    // ---- l0_silu: SILU ----
    v1[0] := v0[0] / (1.0 + EXP(-v0[0]));
    v1[1] := v0[1] / (1.0 + EXP(-v0[1]));
    v1[2] := v0[2] / (1.0 + EXP(-v0[2]));
    v1[3] := v0[3] / (1.0 + EXP(-v0[3]));
    v1[4] := v0[4] / (1.0 + EXP(-v0[4]));
    v1[5] := v0[5] / (1.0 + EXP(-v0[5]));
    v1[6] := v0[6] / (1.0 + EXP(-v0[6]));
    v1[7] := v0[7] / (1.0 + EXP(-v0[7]));
    v1[8] := v0[8] / (1.0 + EXP(-v0[8]));
    v1[9] := v0[9] / (1.0 + EXP(-v0[9]));
    v1[10] := v0[10] / (1.0 + EXP(-v0[10]));
    v1[11] := v0[11] / (1.0 + EXP(-v0[11]));
    v1[12] := v0[12] / (1.0 + EXP(-v0[12]));
    v1[13] := v0[13] / (1.0 + EXP(-v0[13]));
    v1[14] := v0[14] / (1.0 + EXP(-v0[14]));
    v1[15] := v0[15] / (1.0 + EXP(-v0[15]));
    v1[16] := v0[16] / (1.0 + EXP(-v0[16]));
    v1[17] := v0[17] / (1.0 + EXP(-v0[17]));
    v1[18] := v0[18] / (1.0 + EXP(-v0[18]));
    v1[19] := v0[19] / (1.0 + EXP(-v0[19]));
    v1[20] := v0[20] / (1.0 + EXP(-v0[20]));
    v1[21] := v0[21] / (1.0 + EXP(-v0[21]));
    v1[22] := v0[22] / (1.0 + EXP(-v0[22]));
    v1[23] := v0[23] / (1.0 + EXP(-v0[23]));
    v1[24] := v0[24] / (1.0 + EXP(-v0[24]));
    v1[25] := v0[25] / (1.0 + EXP(-v0[25]));
    v1[26] := v0[26] / (1.0 + EXP(-v0[26]));
    v1[27] := v0[27] / (1.0 + EXP(-v0[27]));

    // ---- l0_bspline: BsplineLUT(28x16, 15pts) HOISTED ----
    // Binary search ONCE per input, shared across outputs
    // --- Input 0: binary search ---
    lo := 0; hi := 14;
    WHILE hi - lo > 1 DO
        mid := lo + (hi - lo) / 2;
        IF v0[0] > "NeuroPLC_Weights".w0[mid] THEN lo := mid; ELSE hi := mid; END_IF;
    END_WHILE;
    t_val := (v0[0] - "NeuroPLC_Weights".w0[lo]) / ("NeuroPLC_Weights".w0[hi] - "NeuroPLC_Weights".w0[lo] + 1.0E-10);
    v3[0, 0] := "NeuroPLC_Weights".w1[0 + lo] * (1.0 - t_val) + "NeuroPLC_Weights".w1[0 + hi] * t_val;
    v3[1, 0] := "NeuroPLC_Weights".w1[420 + lo] * (1.0 - t_val) + "NeuroPLC_Weights".w1[420 + hi] * t_val;
    v3[2, 0] := "NeuroPLC_Weights".w1[840 + lo] * (1.0 - t_val) + "NeuroPLC_Weights".w1[840 + hi] * t_val;
    v3[3, 0] := "NeuroPLC_Weights".w1[1260 + lo] * (1.0 - t_val) + "NeuroPLC_Weights".w1[1260 + hi] * t_val;
    v3[4, 0] := "NeuroPLC_Weights".w1[1680 + lo] * (1.0 - t_val) + "NeuroPLC_Weights".w1[1680 + hi] * t_val;
    v3[5, 0] := "NeuroPLC_Weights".w1[2100 + lo] * (1.0 - t_val) + "NeuroPLC_Weights".w1[2100 + hi] * t_val;
    v3[6, 0] := "NeuroPLC_Weights".w1[2520 + lo] * (1.0 - t_val) + "NeuroPLC_Weights".w1[2520 + hi] * t_val;
    v3[7, 0] := "NeuroPLC_Weights".w1[2940 + lo] * (1.0 - t_val) + "NeuroPLC_Weights".w1[2940 + hi] * t_val;
    v3[8, 0] := "NeuroPLC_Weights".w1[3360 + lo] * (1.0 - t_val) + "NeuroPLC_Weights".w1[3360 + hi] * t_val;
    v3[9, 0] := "NeuroPLC_Weights".w1[3780 + lo] * (1.0 - t_val) + "NeuroPLC_Weights".w1[3780 + hi] * t_val;
    v3[10, 0] := "NeuroPLC_Weights".w1[4200 + lo] * (1.0 - t_val) + "NeuroPLC_Weights".w1[4200 + hi] * t_val;
    v3[11, 0] := "NeuroPLC_Weights".w1[4620 + lo] * (1.0 - t_val) + "NeuroPLC_Weights".w1[4620 + hi] * t_val;
    v3[12, 0] := "NeuroPLC_Weights".w1[5040 + lo] * (1.0 - t_val) + "NeuroPLC_Weights".w1[5040 + hi] * t_val;
    v3[13, 0] := "NeuroPLC_Weights".w1[5460 + lo] * (1.0 - t_val) + "NeuroPLC_Weights".w1[5460 + hi] * t_val;
    v3[14, 0] := "NeuroPLC_Weights".w1[5880 + lo] * (1.0 - t_val) + "NeuroPLC_Weights".w1[5880 + hi] * t_val;
    v3[15, 0] := "NeuroPLC_Weights".w1[6300 + lo] * (1.0 - t_val) + "NeuroPLC_Weights".w1[6300 + hi] * t_val;

    // --- Input 1: binary search ---
    lo := 0; hi := 14;
    WHILE hi - lo > 1 DO
        mid := lo + (hi - lo) / 2;
        IF v0[1] > "NeuroPLC_Weights".w0[mid] THEN lo := mid; ELSE hi := mid; END_IF;
    END_WHILE;
    t_val := (v0[1] - "NeuroPLC_Weights".w0[lo]) / ("NeuroPLC_Weights".w0[hi] - "NeuroPLC_Weights".w0[lo] + 1.0E-10);
    v3[0, 1] := "NeuroPLC_Weights".w1[15 + lo] * (1.0 - t_val) + "NeuroPLC_Weights".w1[15 + hi] * t_val;
    v3[1, 1] := "NeuroPLC_Weights".w1[435 + lo] * (1.0 - t_val) + "NeuroPLC_Weights".w1[435 + hi] * t_val;
    v3[2, 1] := "NeuroPLC_Weights".w1[855 + lo] * (1.0 - t_val) + "NeuroPLC_Weights".w1[855 + hi] * t_val;
    v3[3, 1] := "NeuroPLC_Weights".w1[1275 + lo] * (1.0 - t_val) + "NeuroPLC_Weights".w1[1275 + hi] * t_val;
    v3[4, 1] := "NeuroPLC_Weights".w1[1695 + lo] * (1.0 - t_val) + "NeuroPLC_Weights".w1[1695 + hi] * t_val;
    v3[5, 1] := "NeuroPLC_Weights".w1[2115 + lo] * (1.0 - t_val) + "NeuroPLC_Weights".w1[2115 + hi] * t_val;
    v3[6, 1] := "NeuroPLC_Weights".w1[2535 + lo] * (1.0 - t_val) + "NeuroPLC_Weights".w1[2535 + hi] * t_val;
    v3[7, 1] := "NeuroPLC_Weights".w1[2955 + lo] * (1.0 - t_val) + "NeuroPLC_Weights".w1[2955 + hi] * t_val;
    v3[8, 1] := "NeuroPLC_Weights".w1[3375 + lo] * (1.0 - t_val) + "NeuroPLC_Weights".w1[3375 + hi] * t_val;
    v3[9, 1] := "NeuroPLC_Weights".w1[3795 + lo] * (1.0 - t_val) + "NeuroPLC_Weights".w1[3795 + hi] * t_val;
    v3[10, 1] := "NeuroPLC_Weights".w1[4215 + lo] * (1.0 - t_val) + "NeuroPLC_Weights".w1[4215 + hi] * t_val;
    v3[11, 1] := "NeuroPLC_Weights".w1[4635 + lo] * (1.0 - t_val) + "NeuroPLC_Weights".w1[4635 + hi] * t_val;
    v3[12, 1] := "NeuroPLC_Weights".w1[5055 + lo] * (1.0 - t_val) + "NeuroPLC_Weights".w1[5055 + hi] * t_val;
    v3[13, 1] := "NeuroPLC_Weights".w1[5475 + lo] * (1.0 - t_val) + "NeuroPLC_Weights".w1[5475 + hi] * t_val;
    v3[14, 1] := "NeuroPLC_Weights".w1[5895 + lo] * (1.0 - t_val) + "NeuroPLC_Weights".w1[5895 + hi] * t_val;
    v3[15, 1] := "NeuroPLC_Weights".w1[6315 + lo] * (1.0 - t_val) + "NeuroPLC_Weights".w1[6315 + hi] * t_val;

    // --- Input 2: binary search ---
    lo := 0; hi := 14;
    WHILE hi - lo > 1 DO
        mid := lo + (hi - lo) / 2;
        IF v0[2] > "NeuroPLC_Weights".w0[mid] THEN lo := mid; ELSE hi := mid; END_IF;
    END_WHILE;
    t_val := (v0[2] - "NeuroPLC_Weights".w0[lo]) / ("NeuroPLC_Weights".w0[hi] - "NeuroPLC_Weights".w0[lo] + 1.0E-10);
    v3[0, 2] := "NeuroPLC_Weights".w1[30 + lo] * (1.0 - t_val) + "NeuroPLC_Weights".w1[30 + hi] * t_val;
    v3[1, 2] := "NeuroPLC_Weights".w1[450 + lo] * (1.0 - t_val) + "NeuroPLC_Weights".w1[450 + hi] * t_val;
    v3[2, 2] := "NeuroPLC_Weights".w1[870 + lo] * (1.0 - t_val) + "NeuroPLC_Weights".w1[870 + hi] * t_val;
    v3[3, 2] := "NeuroPLC_Weights".w1[1290 + lo] * (1.0 - t_val) + "NeuroPLC_Weights".w1[1290 + hi] * t_val;
    v3[4, 2] := "NeuroPLC_Weights".w1[1710 + lo] * (1.0 - t_val) + "NeuroPLC_Weights".w1[1710 + hi] * t_val;
    v3[5, 2] := "NeuroPLC_Weights".w1[2130 + lo] * (1.0 - t_val) + "NeuroPLC_Weights".w1[2130 + hi] * t_val;
    v3[6, 2] := "NeuroPLC_Weights".w1[2550 + lo] * (1.0 - t_val) + "NeuroPLC_Weights".w1[2550 + hi] * t_val;
    v3[7, 2] := "NeuroPLC_Weights".w1[2970 + lo] * (1.0 - t_val) + "NeuroPLC_Weights".w1[2970 + hi] * t_val;
    v3[8, 2] := "NeuroPLC_Weights".w1[3390 + lo] * (1.0 - t_val) + "NeuroPLC_Weights".w1[3390 + hi] * t_val;
    v3[9, 2] := "NeuroPLC_Weights".w1[3810 + lo] * (1.0 - t_val) + "NeuroPLC_Weights".w1[3810 + hi] * t_val;
    v3[10, 2] := "NeuroPLC_Weights".w1[4230 + lo] * (1.0 - t_val) + "NeuroPLC_Weights".w1[4230 + hi] * t_val;
    v3[11, 2] := "NeuroPLC_Weights".w1[4650 + lo] * (1.0 - t_val) + "NeuroPLC_Weights".w1[4650 + hi] * t_val;
    v3[12, 2] := "NeuroPLC_Weights".w1[5070 + lo] * (1.0 - t_val) + "NeuroPLC_Weights".w1[5070 + hi] * t_val;
    v3[13, 2] := "NeuroPLC_Weights".w1[5490 + lo] * (1.0 - t_val) + "NeuroPLC_Weights".w1[5490 + hi] * t_val;
    v3[14, 2] := "NeuroPLC_Weights".w1[5910 + lo] * (1.0 - t_val) + "NeuroPLC_Weights".w1[5910 + hi] * t_val;
    v3[15, 2] := "NeuroPLC_Weights".w1[6330 + lo] * (1.0 - t_val) + "NeuroPLC_Weights".w1[6330 + hi] * t_val;

    // --- Input 3: binary search ---
    lo := 0; hi := 14;
    WHILE hi - lo > 1 DO
        mid := lo + (hi - lo) / 2;
        IF v0[3] > "NeuroPLC_Weights".w0[mid] THEN lo := mid; ELSE hi := mid; END_IF;
    END_WHILE;
    t_val := (v0[3] - "NeuroPLC_Weights".w0[lo]) / ("NeuroPLC_Weights".w0[hi] - "NeuroPLC_Weights".w0[lo] + 1.0E-10);
    v3[0, 3] := "NeuroPLC_Weights".w1[45 + lo] * (1.0 - t_val) + "NeuroPLC_Weights".w1[45 + hi] * t_val;
    v3[1, 3] := "NeuroPLC_Weights".w1[465 + lo] * (1.0 - t_val) + "NeuroPLC_Weights".w1[465 + hi] * t_val;
    v3[2, 3] := "NeuroPLC_Weights".w1[885 + lo] * (1.0 - t_val) + "NeuroPLC_Weights".w1[885 + hi] * t_val;
    v3[3, 3] := "NeuroPLC_Weights".w1[1305 + lo] * (1.0 - t_val) + "NeuroPLC_Weights".w1[1305 + hi] * t_val;
    v3[4, 3] := "NeuroPLC_Weights".w1[1725 + lo] * (1.0 - t_val) + "NeuroPLC_Weights".w1[1725 + hi] * t_val;
    v3[5, 3] := "NeuroPLC_Weights".w1[2145 + lo] * (1.0 - t_val) + "NeuroPLC_Weights".w1[2145 + hi] * t_val;
    v3[6, 3] := "NeuroPLC_Weights".w1[2565 + lo] * (1.0 - t_val) + "NeuroPLC_Weights".w1[2565 + hi] * t_val;
    v3[7, 3] := "NeuroPLC_Weights".w1[2985 + lo] * (1.0 - t_val) + "NeuroPLC_Weights".w1[2985 + hi] * t_val;
    v3[8, 3] := "NeuroPLC_Weights".w1[3405 + lo] * (1.0 - t_val) + "NeuroPLC_Weights".w1[3405 + hi] * t_val;
    v3[9, 3] := "NeuroPLC_Weights".w1[3825 + lo] * (1.0 - t_val) + "NeuroPLC_Weights".w1[3825 + hi] * t_val;
    v3[10, 3] := "NeuroPLC_Weights".w1[4245 + lo] * (1.0 - t_val) + "NeuroPLC_Weights".w1[4245 + hi] * t_val;
    v3[11, 3] := "NeuroPLC_Weights".w1[4665 + lo] * (1.0 - t_val) + "NeuroPLC_Weights".w1[4665 + hi] * t_val;
    v3[12, 3] := "NeuroPLC_Weights".w1[5085 + lo] * (1.0 - t_val) + "NeuroPLC_Weights".w1[5085 + hi] * t_val;
    v3[13, 3] := "NeuroPLC_Weights".w1[5505 + lo] * (1.0 - t_val) + "NeuroPLC_Weights".w1[5505 + hi] * t_val;
    v3[14, 3] := "NeuroPLC_Weights".w1[5925 + lo] * (1.0 - t_val) + "NeuroPLC_Weights".w1[5925 + hi] * t_val;
    v3[15, 3] := "NeuroPLC_Weights".w1[6345 + lo] * (1.0 - t_val) + "NeuroPLC_Weights".w1[6345 + hi] * t_val;

    // --- Input 4: binary search ---
    lo := 0; hi := 14;
    WHILE hi - lo > 1 DO
        mid := lo + (hi - lo) / 2;
        IF v0[4] > "NeuroPLC_Weights".w0[mid] THEN lo := mid; ELSE hi := mid; END_IF;
    END_WHILE;
    t_val := (v0[4] - "NeuroPLC_Weights".w0[lo]) / ("NeuroPLC_Weights".w0[hi] - "NeuroPLC_Weights".w0[lo] + 1.0E-10);
    v3[0, 4] := "NeuroPLC_Weights".w1[60 + lo] * (1.0 - t_val) + "NeuroPLC_Weights".w1[60 + hi] * t_val;
    v3[1, 4] := "NeuroPLC_Weights".w1[480 + lo] * (1.0 - t_val) + "NeuroPLC_Weights".w1[480 + hi] * t_val;
    v3[2, 4] := "NeuroPLC_Weights".w1[900 + lo] * (1.0 - t_val) + "NeuroPLC_Weights".w1[900 + hi] * t_val;
    v3[3, 4] := "NeuroPLC_Weights".w1[1320 + lo] * (1.0 - t_val) + "NeuroPLC_Weights".w1[1320 + hi] * t_val;
    v3[4, 4] := "NeuroPLC_Weights".w1[1740 + lo] * (1.0 - t_val) + "NeuroPLC_Weights".w1[1740 + hi] * t_val;
    v3[5, 4] := "NeuroPLC_Weights".w1[2160 + lo] * (1.0 - t_val) + "NeuroPLC_Weights".w1[2160 + hi] * t_val;
    v3[6, 4] := "NeuroPLC_Weights".w1[2580 + lo] * (1.0 - t_val) + "NeuroPLC_Weights".w1[2580 + hi] * t_val;
    v3[7, 4] := "NeuroPLC_Weights".w1[3000 + lo] * (1.0 - t_val) + "NeuroPLC_Weights".w1[3000 + hi] * t_val;
    v3[8, 4] := "NeuroPLC_Weights".w1[3420 + lo] * (1.0 - t_val) + "NeuroPLC_Weights".w1[3420 + hi] * t_val;
    v3[9, 4] := "NeuroPLC_Weights".w1[3840 + lo] * (1.0 - t_val) + "NeuroPLC_Weights".w1[3840 + hi] * t_val;
    v3[10, 4] := "NeuroPLC_Weights".w1[4260 + lo] * (1.0 - t_val) + "NeuroPLC_Weights".w1[4260 + hi] * t_val;
    v3[11, 4] := "NeuroPLC_Weights".w1[4680 + lo] * (1.0 - t_val) + "NeuroPLC_Weights".w1[4680 + hi] * t_val;
    v3[12, 4] := "NeuroPLC_Weights".w1[5100 + lo] * (1.0 - t_val) + "NeuroPLC_Weights".w1[5100 + hi] * t_val;
    v3[13, 4] := "NeuroPLC_Weights".w1[5520 + lo] * (1.0 - t_val) + "NeuroPLC_Weights".w1[5520 + hi] * t_val;
    v3[14, 4] := "NeuroPLC_Weights".w1[5940 + lo] * (1.0 - t_val) + "NeuroPLC_Weights".w1[5940 + hi] * t_val;
    v3[15, 4] := "NeuroPLC_Weights".w1[6360 + lo] * (1.0 - t_val) + "NeuroPLC_Weights".w1[6360 + hi] * t_val;

    // --- Input 5: binary search ---
    lo := 0; hi := 14;
    WHILE hi - lo > 1 DO
        mid := lo + (hi - lo) / 2;
        IF v0[5] > "NeuroPLC_Weights".w0[mid] THEN lo := mid; ELSE hi := mid; END_IF;
    END_WHILE;
    t_val := (v0[5] - "NeuroPLC_Weights".w0[lo]) / ("NeuroPLC_Weights".w0[hi] - "NeuroPLC_Weights".w0[lo] + 1.0E-10);
    v3[0, 5] := "NeuroPLC_Weights".w1[75 + lo] * (1.0 - t_val) + "NeuroPLC_Weights".w1[75 + hi] * t_val;
    v3[1, 5] := "NeuroPLC_Weights".w1[495 + lo] * (1.0 - t_val) + "NeuroPLC_Weights".w1[495 + hi] * t_val;
    v3[2, 5] := "NeuroPLC_Weights".w1[915 + lo] * (1.0 - t_val) + "NeuroPLC_Weights".w1[915 + hi] * t_val;
    v3[3, 5] := "NeuroPLC_Weights".w1[1335 + lo] * (1.0 - t_val) + "NeuroPLC_Weights".w1[1335 + hi] * t_val;
    v3[4, 5] := "NeuroPLC_Weights".w1[1755 + lo] * (1.0 - t_val) + "NeuroPLC_Weights".w1[1755 + hi] * t_val;
    v3[5, 5] := "NeuroPLC_Weights".w1[2175 + lo] * (1.0 - t_val) + "NeuroPLC_Weights".w1[2175 + hi] * t_val;
    v3[6, 5] := "NeuroPLC_Weights".w1[2595 + lo] * (1.0 - t_val) + "NeuroPLC_Weights".w1[2595 + hi] * t_val;
    v3[7, 5] := "NeuroPLC_Weights".w1[3015 + lo] * (1.0 - t_val) + "NeuroPLC_Weights".w1[3015 + hi] * t_val;
    v3[8, 5] := "NeuroPLC_Weights".w1[3435 + lo] * (1.0 - t_val) + "NeuroPLC_Weights".w1[3435 + hi] * t_val;
    v3[9, 5] := "NeuroPLC_Weights".w1[3855 + lo] * (1.0 - t_val) + "NeuroPLC_Weights".w1[3855 + hi] * t_val;
    v3[10, 5] := "NeuroPLC_Weights".w1[4275 + lo] * (1.0 - t_val) + "NeuroPLC_Weights".w1[4275 + hi] * t_val;
    v3[11, 5] := "NeuroPLC_Weights".w1[4695 + lo] * (1.0 - t_val) + "NeuroPLC_Weights".w1[4695 + hi] * t_val;
    v3[12, 5] := "NeuroPLC_Weights".w1[5115 + lo] * (1.0 - t_val) + "NeuroPLC_Weights".w1[5115 + hi] * t_val;
    v3[13, 5] := "NeuroPLC_Weights".w1[5535 + lo] * (1.0 - t_val) + "NeuroPLC_Weights".w1[5535 + hi] * t_val;
    v3[14, 5] := "NeuroPLC_Weights".w1[5955 + lo] * (1.0 - t_val) + "NeuroPLC_Weights".w1[5955 + hi] * t_val;
    v3[15, 5] := "NeuroPLC_Weights".w1[6375 + lo] * (1.0 - t_val) + "NeuroPLC_Weights".w1[6375 + hi] * t_val;

    // --- Input 6: binary search ---
    lo := 0; hi := 14;
    WHILE hi - lo > 1 DO
        mid := lo + (hi - lo) / 2;
        IF v0[6] > "NeuroPLC_Weights".w0[mid] THEN lo := mid; ELSE hi := mid; END_IF;
    END_WHILE;
    t_val := (v0[6] - "NeuroPLC_Weights".w0[lo]) / ("NeuroPLC_Weights".w0[hi] - "NeuroPLC_Weights".w0[lo] + 1.0E-10);
    v3[0, 6] := "NeuroPLC_Weights".w1[90 + lo] * (1.0 - t_val) + "NeuroPLC_Weights".w1[90 + hi] * t_val;
    v3[1, 6] := "NeuroPLC_Weights".w1[510 + lo] * (1.0 - t_val) + "NeuroPLC_Weights".w1[510 + hi] * t_val;
    v3[2, 6] := "NeuroPLC_Weights".w1[930 + lo] * (1.0 - t_val) + "NeuroPLC_Weights".w1[930 + hi] * t_val;
    v3[3, 6] := "NeuroPLC_Weights".w1[1350 + lo] * (1.0 - t_val) + "NeuroPLC_Weights".w1[1350 + hi] * t_val;
    v3[4, 6] := "NeuroPLC_Weights".w1[1770 + lo] * (1.0 - t_val) + "NeuroPLC_Weights".w1[1770 + hi] * t_val;
    v3[5, 6] := "NeuroPLC_Weights".w1[2190 + lo] * (1.0 - t_val) + "NeuroPLC_Weights".w1[2190 + hi] * t_val;
    v3[6, 6] := "NeuroPLC_Weights".w1[2610 + lo] * (1.0 - t_val) + "NeuroPLC_Weights".w1[2610 + hi] * t_val;
    v3[7, 6] := "NeuroPLC_Weights".w1[3030 + lo] * (1.0 - t_val) + "NeuroPLC_Weights".w1[3030 + hi] * t_val;
    v3[8, 6] := "NeuroPLC_Weights".w1[3450 + lo] * (1.0 - t_val) + "NeuroPLC_Weights".w1[3450 + hi] * t_val;
    v3[9, 6] := "NeuroPLC_Weights".w1[3870 + lo] * (1.0 - t_val) + "NeuroPLC_Weights".w1[3870 + hi] * t_val;
    v3[10, 6] := "NeuroPLC_Weights".w1[4290 + lo] * (1.0 - t_val) + "NeuroPLC_Weights".w1[4290 + hi] * t_val;
    v3[11, 6] := "NeuroPLC_Weights".w1[4710 + lo] * (1.0 - t_val) + "NeuroPLC_Weights".w1[4710 + hi] * t_val;
    v3[12, 6] := "NeuroPLC_Weights".w1[5130 + lo] * (1.0 - t_val) + "NeuroPLC_Weights".w1[5130 + hi] * t_val;
    v3[13, 6] := "NeuroPLC_Weights".w1[5550 + lo] * (1.0 - t_val) + "NeuroPLC_Weights".w1[5550 + hi] * t_val;
    v3[14, 6] := "NeuroPLC_Weights".w1[5970 + lo] * (1.0 - t_val) + "NeuroPLC_Weights".w1[5970 + hi] * t_val;
    v3[15, 6] := "NeuroPLC_Weights".w1[6390 + lo] * (1.0 - t_val) + "NeuroPLC_Weights".w1[6390 + hi] * t_val;

    // --- Input 7: binary search ---
    lo := 0; hi := 14;
    WHILE hi - lo > 1 DO
        mid := lo + (hi - lo) / 2;
        IF v0[7] > "NeuroPLC_Weights".w0[mid] THEN lo := mid; ELSE hi := mid; END_IF;
    END_WHILE;
    t_val := (v0[7] - "NeuroPLC_Weights".w0[lo]) / ("NeuroPLC_Weights".w0[hi] - "NeuroPLC_Weights".w0[lo] + 1.0E-10);
    v3[0, 7] := "NeuroPLC_Weights".w1[105 + lo] * (1.0 - t_val) + "NeuroPLC_Weights".w1[105 + hi] * t_val;
    v3[1, 7] := "NeuroPLC_Weights".w1[525 + lo] * (1.0 - t_val) + "NeuroPLC_Weights".w1[525 + hi] * t_val;
    v3[2, 7] := "NeuroPLC_Weights".w1[945 + lo] * (1.0 - t_val) + "NeuroPLC_Weights".w1[945 + hi] * t_val;
    v3[3, 7] := "NeuroPLC_Weights".w1[1365 + lo] * (1.0 - t_val) + "NeuroPLC_Weights".w1[1365 + hi] * t_val;
    v3[4, 7] := "NeuroPLC_Weights".w1[1785 + lo] * (1.0 - t_val) + "NeuroPLC_Weights".w1[1785 + hi] * t_val;
    v3[5, 7] := "NeuroPLC_Weights".w1[2205 + lo] * (1.0 - t_val) + "NeuroPLC_Weights".w1[2205 + hi] * t_val;
    v3[6, 7] := "NeuroPLC_Weights".w1[2625 + lo] * (1.0 - t_val) + "NeuroPLC_Weights".w1[2625 + hi] * t_val;
    v3[7, 7] := "NeuroPLC_Weights".w1[3045 + lo] * (1.0 - t_val) + "NeuroPLC_Weights".w1[3045 + hi] * t_val;
    v3[8, 7] := "NeuroPLC_Weights".w1[3465 + lo] * (1.0 - t_val) + "NeuroPLC_Weights".w1[3465 + hi] * t_val;
    v3[9, 7] := "NeuroPLC_Weights".w1[3885 + lo] * (1.0 - t_val) + "NeuroPLC_Weights".w1[3885 + hi] * t_val;
    v3[10, 7] := "NeuroPLC_Weights".w1[4305 + lo] * (1.0 - t_val) + "NeuroPLC_Weights".w1[4305 + hi] * t_val;
    v3[11, 7] := "NeuroPLC_Weights".w1[4725 + lo] * (1.0 - t_val) + "NeuroPLC_Weights".w1[4725 + hi] * t_val;
    v3[12, 7] := "NeuroPLC_Weights".w1[5145 + lo] * (1.0 - t_val) + "NeuroPLC_Weights".w1[5145 + hi] * t_val;
    v3[13, 7] := "NeuroPLC_Weights".w1[5565 + lo] * (1.0 - t_val) + "NeuroPLC_Weights".w1[5565 + hi] * t_val;
    v3[14, 7] := "NeuroPLC_Weights".w1[5985 + lo] * (1.0 - t_val) + "NeuroPLC_Weights".w1[5985 + hi] * t_val;
    v3[15, 7] := "NeuroPLC_Weights".w1[6405 + lo] * (1.0 - t_val) + "NeuroPLC_Weights".w1[6405 + hi] * t_val;

    // --- Input 8: binary search ---
    lo := 0; hi := 14;
    WHILE hi - lo > 1 DO
        mid := lo + (hi - lo) / 2;
        IF v0[8] > "NeuroPLC_Weights".w0[mid] THEN lo := mid; ELSE hi := mid; END_IF;
    END_WHILE;
    t_val := (v0[8] - "NeuroPLC_Weights".w0[lo]) / ("NeuroPLC_Weights".w0[hi] - "NeuroPLC_Weights".w0[lo] + 1.0E-10);
    v3[0, 8] := "NeuroPLC_Weights".w1[120 + lo] * (1.0 - t_val) + "NeuroPLC_Weights".w1[120 + hi] * t_val;
    v3[1, 8] := "NeuroPLC_Weights".w1[540 + lo] * (1.0 - t_val) + "NeuroPLC_Weights".w1[540 + hi] * t_val;
    v3[2, 8] := "NeuroPLC_Weights".w1[960 + lo] * (1.0 - t_val) + "NeuroPLC_Weights".w1[960 + hi] * t_val;
    v3[3, 8] := "NeuroPLC_Weights".w1[1380 + lo] * (1.0 - t_val) + "NeuroPLC_Weights".w1[1380 + hi] * t_val;
    v3[4, 8] := "NeuroPLC_Weights".w1[1800 + lo] * (1.0 - t_val) + "NeuroPLC_Weights".w1[1800 + hi] * t_val;
    v3[5, 8] := "NeuroPLC_Weights".w1[2220 + lo] * (1.0 - t_val) + "NeuroPLC_Weights".w1[2220 + hi] * t_val;
    v3[6, 8] := "NeuroPLC_Weights".w1[2640 + lo] * (1.0 - t_val) + "NeuroPLC_Weights".w1[2640 + hi] * t_val;
    v3[7, 8] := "NeuroPLC_Weights".w1[3060 + lo] * (1.0 - t_val) + "NeuroPLC_Weights".w1[3060 + hi] * t_val;
    v3[8, 8] := "NeuroPLC_Weights".w1[3480 + lo] * (1.0 - t_val) + "NeuroPLC_Weights".w1[3480 + hi] * t_val;
    v3[9, 8] := "NeuroPLC_Weights".w1[3900 + lo] * (1.0 - t_val) + "NeuroPLC_Weights".w1[3900 + hi] * t_val;
    v3[10, 8] := "NeuroPLC_Weights".w1[4320 + lo] * (1.0 - t_val) + "NeuroPLC_Weights".w1[4320 + hi] * t_val;
    v3[11, 8] := "NeuroPLC_Weights".w1[4740 + lo] * (1.0 - t_val) + "NeuroPLC_Weights".w1[4740 + hi] * t_val;
    v3[12, 8] := "NeuroPLC_Weights".w1[5160 + lo] * (1.0 - t_val) + "NeuroPLC_Weights".w1[5160 + hi] * t_val;
    v3[13, 8] := "NeuroPLC_Weights".w1[5580 + lo] * (1.0 - t_val) + "NeuroPLC_Weights".w1[5580 + hi] * t_val;
    v3[14, 8] := "NeuroPLC_Weights".w1[6000 + lo] * (1.0 - t_val) + "NeuroPLC_Weights".w1[6000 + hi] * t_val;
    v3[15, 8] := "NeuroPLC_Weights".w1[6420 + lo] * (1.0 - t_val) + "NeuroPLC_Weights".w1[6420 + hi] * t_val;

    // --- Input 9: binary search ---
    lo := 0; hi := 14;
    WHILE hi - lo > 1 DO
        mid := lo + (hi - lo) / 2;
        IF v0[9] > "NeuroPLC_Weights".w0[mid] THEN lo := mid; ELSE hi := mid; END_IF;
    END_WHILE;
    t_val := (v0[9] - "NeuroPLC_Weights".w0[lo]) / ("NeuroPLC_Weights".w0[hi] - "NeuroPLC_Weights".w0[lo] + 1.0E-10);
    v3[0, 9] := "NeuroPLC_Weights".w1[135 + lo] * (1.0 - t_val) + "NeuroPLC_Weights".w1[135 + hi] * t_val;
    v3[1, 9] := "NeuroPLC_Weights".w1[555 + lo] * (1.0 - t_val) + "NeuroPLC_Weights".w1[555 + hi] * t_val;
    v3[2, 9] := "NeuroPLC_Weights".w1[975 + lo] * (1.0 - t_val) + "NeuroPLC_Weights".w1[975 + hi] * t_val;
    v3[3, 9] := "NeuroPLC_Weights".w1[1395 + lo] * (1.0 - t_val) + "NeuroPLC_Weights".w1[1395 + hi] * t_val;
    v3[4, 9] := "NeuroPLC_Weights".w1[1815 + lo] * (1.0 - t_val) + "NeuroPLC_Weights".w1[1815 + hi] * t_val;
    v3[5, 9] := "NeuroPLC_Weights".w1[2235 + lo] * (1.0 - t_val) + "NeuroPLC_Weights".w1[2235 + hi] * t_val;
    v3[6, 9] := "NeuroPLC_Weights".w1[2655 + lo] * (1.0 - t_val) + "NeuroPLC_Weights".w1[2655 + hi] * t_val;
    v3[7, 9] := "NeuroPLC_Weights".w1[3075 + lo] * (1.0 - t_val) + "NeuroPLC_Weights".w1[3075 + hi] * t_val;
    v3[8, 9] := "NeuroPLC_Weights".w1[3495 + lo] * (1.0 - t_val) + "NeuroPLC_Weights".w1[3495 + hi] * t_val;
    v3[9, 9] := "NeuroPLC_Weights".w1[3915 + lo] * (1.0 - t_val) + "NeuroPLC_Weights".w1[3915 + hi] * t_val;
    v3[10, 9] := "NeuroPLC_Weights".w1[4335 + lo] * (1.0 - t_val) + "NeuroPLC_Weights".w1[4335 + hi] * t_val;
    v3[11, 9] := "NeuroPLC_Weights".w1[4755 + lo] * (1.0 - t_val) + "NeuroPLC_Weights".w1[4755 + hi] * t_val;
    v3[12, 9] := "NeuroPLC_Weights".w1[5175 + lo] * (1.0 - t_val) + "NeuroPLC_Weights".w1[5175 + hi] * t_val;
    v3[13, 9] := "NeuroPLC_Weights".w1[5595 + lo] * (1.0 - t_val) + "NeuroPLC_Weights".w1[5595 + hi] * t_val;
    v3[14, 9] := "NeuroPLC_Weights".w1[6015 + lo] * (1.0 - t_val) + "NeuroPLC_Weights".w1[6015 + hi] * t_val;
    v3[15, 9] := "NeuroPLC_Weights".w1[6435 + lo] * (1.0 - t_val) + "NeuroPLC_Weights".w1[6435 + hi] * t_val;

    // --- Input 10: binary search ---
    lo := 0; hi := 14;
    WHILE hi - lo > 1 DO
        mid := lo + (hi - lo) / 2;
        IF v0[10] > "NeuroPLC_Weights".w0[mid] THEN lo := mid; ELSE hi := mid; END_IF;
    END_WHILE;
    t_val := (v0[10] - "NeuroPLC_Weights".w0[lo]) / ("NeuroPLC_Weights".w0[hi] - "NeuroPLC_Weights".w0[lo] + 1.0E-10);
    v3[0, 10] := "NeuroPLC_Weights".w1[150 + lo] * (1.0 - t_val) + "NeuroPLC_Weights".w1[150 + hi] * t_val;
    v3[1, 10] := "NeuroPLC_Weights".w1[570 + lo] * (1.0 - t_val) + "NeuroPLC_Weights".w1[570 + hi] * t_val;
    v3[2, 10] := "NeuroPLC_Weights".w1[990 + lo] * (1.0 - t_val) + "NeuroPLC_Weights".w1[990 + hi] * t_val;
    v3[3, 10] := "NeuroPLC_Weights".w1[1410 + lo] * (1.0 - t_val) + "NeuroPLC_Weights".w1[1410 + hi] * t_val;
    v3[4, 10] := "NeuroPLC_Weights".w1[1830 + lo] * (1.0 - t_val) + "NeuroPLC_Weights".w1[1830 + hi] * t_val;
    v3[5, 10] := "NeuroPLC_Weights".w1[2250 + lo] * (1.0 - t_val) + "NeuroPLC_Weights".w1[2250 + hi] * t_val;
    v3[6, 10] := "NeuroPLC_Weights".w1[2670 + lo] * (1.0 - t_val) + "NeuroPLC_Weights".w1[2670 + hi] * t_val;
    v3[7, 10] := "NeuroPLC_Weights".w1[3090 + lo] * (1.0 - t_val) + "NeuroPLC_Weights".w1[3090 + hi] * t_val;
    v3[8, 10] := "NeuroPLC_Weights".w1[3510 + lo] * (1.0 - t_val) + "NeuroPLC_Weights".w1[3510 + hi] * t_val;
    v3[9, 10] := "NeuroPLC_Weights".w1[3930 + lo] * (1.0 - t_val) + "NeuroPLC_Weights".w1[3930 + hi] * t_val;
    v3[10, 10] := "NeuroPLC_Weights".w1[4350 + lo] * (1.0 - t_val) + "NeuroPLC_Weights".w1[4350 + hi] * t_val;
    v3[11, 10] := "NeuroPLC_Weights".w1[4770 + lo] * (1.0 - t_val) + "NeuroPLC_Weights".w1[4770 + hi] * t_val;
    v3[12, 10] := "NeuroPLC_Weights".w1[5190 + lo] * (1.0 - t_val) + "NeuroPLC_Weights".w1[5190 + hi] * t_val;
    v3[13, 10] := "NeuroPLC_Weights".w1[5610 + lo] * (1.0 - t_val) + "NeuroPLC_Weights".w1[5610 + hi] * t_val;
    v3[14, 10] := "NeuroPLC_Weights".w1[6030 + lo] * (1.0 - t_val) + "NeuroPLC_Weights".w1[6030 + hi] * t_val;
    v3[15, 10] := "NeuroPLC_Weights".w1[6450 + lo] * (1.0 - t_val) + "NeuroPLC_Weights".w1[6450 + hi] * t_val;

    // --- Input 11: binary search ---
    lo := 0; hi := 14;
    WHILE hi - lo > 1 DO
        mid := lo + (hi - lo) / 2;
        IF v0[11] > "NeuroPLC_Weights".w0[mid] THEN lo := mid; ELSE hi := mid; END_IF;
    END_WHILE;
    t_val := (v0[11] - "NeuroPLC_Weights".w0[lo]) / ("NeuroPLC_Weights".w0[hi] - "NeuroPLC_Weights".w0[lo] + 1.0E-10);
    v3[0, 11] := "NeuroPLC_Weights".w1[165 + lo] * (1.0 - t_val) + "NeuroPLC_Weights".w1[165 + hi] * t_val;
    v3[1, 11] := "NeuroPLC_Weights".w1[585 + lo] * (1.0 - t_val) + "NeuroPLC_Weights".w1[585 + hi] * t_val;
    v3[2, 11] := "NeuroPLC_Weights".w1[1005 + lo] * (1.0 - t_val) + "NeuroPLC_Weights".w1[1005 + hi] * t_val;
    v3[3, 11] := "NeuroPLC_Weights".w1[1425 + lo] * (1.0 - t_val) + "NeuroPLC_Weights".w1[1425 + hi] * t_val;
    v3[4, 11] := "NeuroPLC_Weights".w1[1845 + lo] * (1.0 - t_val) + "NeuroPLC_Weights".w1[1845 + hi] * t_val;
    v3[5, 11] := "NeuroPLC_Weights".w1[2265 + lo] * (1.0 - t_val) + "NeuroPLC_Weights".w1[2265 + hi] * t_val;
    v3[6, 11] := "NeuroPLC_Weights".w1[2685 + lo] * (1.0 - t_val) + "NeuroPLC_Weights".w1[2685 + hi] * t_val;
    v3[7, 11] := "NeuroPLC_Weights".w1[3105 + lo] * (1.0 - t_val) + "NeuroPLC_Weights".w1[3105 + hi] * t_val;
    v3[8, 11] := "NeuroPLC_Weights".w1[3525 + lo] * (1.0 - t_val) + "NeuroPLC_Weights".w1[3525 + hi] * t_val;
    v3[9, 11] := "NeuroPLC_Weights".w1[3945 + lo] * (1.0 - t_val) + "NeuroPLC_Weights".w1[3945 + hi] * t_val;
    v3[10, 11] := "NeuroPLC_Weights".w1[4365 + lo] * (1.0 - t_val) + "NeuroPLC_Weights".w1[4365 + hi] * t_val;
    v3[11, 11] := "NeuroPLC_Weights".w1[4785 + lo] * (1.0 - t_val) + "NeuroPLC_Weights".w1[4785 + hi] * t_val;
    v3[12, 11] := "NeuroPLC_Weights".w1[5205 + lo] * (1.0 - t_val) + "NeuroPLC_Weights".w1[5205 + hi] * t_val;
    v3[13, 11] := "NeuroPLC_Weights".w1[5625 + lo] * (1.0 - t_val) + "NeuroPLC_Weights".w1[5625 + hi] * t_val;
    v3[14, 11] := "NeuroPLC_Weights".w1[6045 + lo] * (1.0 - t_val) + "NeuroPLC_Weights".w1[6045 + hi] * t_val;
    v3[15, 11] := "NeuroPLC_Weights".w1[6465 + lo] * (1.0 - t_val) + "NeuroPLC_Weights".w1[6465 + hi] * t_val;

    // --- Input 12: binary search ---
    lo := 0; hi := 14;
    WHILE hi - lo > 1 DO
        mid := lo + (hi - lo) / 2;
        IF v0[12] > "NeuroPLC_Weights".w0[mid] THEN lo := mid; ELSE hi := mid; END_IF;
    END_WHILE;
    t_val := (v0[12] - "NeuroPLC_Weights".w0[lo]) / ("NeuroPLC_Weights".w0[hi] - "NeuroPLC_Weights".w0[lo] + 1.0E-10);
    v3[0, 12] := "NeuroPLC_Weights".w1[180 + lo] * (1.0 - t_val) + "NeuroPLC_Weights".w1[180 + hi] * t_val;
    v3[1, 12] := "NeuroPLC_Weights".w1[600 + lo] * (1.0 - t_val) + "NeuroPLC_Weights".w1[600 + hi] * t_val;
    v3[2, 12] := "NeuroPLC_Weights".w1[1020 + lo] * (1.0 - t_val) + "NeuroPLC_Weights".w1[1020 + hi] * t_val;
    v3[3, 12] := "NeuroPLC_Weights".w1[1440 + lo] * (1.0 - t_val) + "NeuroPLC_Weights".w1[1440 + hi] * t_val;
    v3[4, 12] := "NeuroPLC_Weights".w1[1860 + lo] * (1.0 - t_val) + "NeuroPLC_Weights".w1[1860 + hi] * t_val;
    v3[5, 12] := "NeuroPLC_Weights".w1[2280 + lo] * (1.0 - t_val) + "NeuroPLC_Weights".w1[2280 + hi] * t_val;
    v3[6, 12] := "NeuroPLC_Weights".w1[2700 + lo] * (1.0 - t_val) + "NeuroPLC_Weights".w1[2700 + hi] * t_val;
    v3[7, 12] := "NeuroPLC_Weights".w1[3120 + lo] * (1.0 - t_val) + "NeuroPLC_Weights".w1[3120 + hi] * t_val;
    v3[8, 12] := "NeuroPLC_Weights".w1[3540 + lo] * (1.0 - t_val) + "NeuroPLC_Weights".w1[3540 + hi] * t_val;
    v3[9, 12] := "NeuroPLC_Weights".w1[3960 + lo] * (1.0 - t_val) + "NeuroPLC_Weights".w1[3960 + hi] * t_val;
    v3[10, 12] := "NeuroPLC_Weights".w1[4380 + lo] * (1.0 - t_val) + "NeuroPLC_Weights".w1[4380 + hi] * t_val;
    v3[11, 12] := "NeuroPLC_Weights".w1[4800 + lo] * (1.0 - t_val) + "NeuroPLC_Weights".w1[4800 + hi] * t_val;
    v3[12, 12] := "NeuroPLC_Weights".w1[5220 + lo] * (1.0 - t_val) + "NeuroPLC_Weights".w1[5220 + hi] * t_val;
    v3[13, 12] := "NeuroPLC_Weights".w1[5640 + lo] * (1.0 - t_val) + "NeuroPLC_Weights".w1[5640 + hi] * t_val;
    v3[14, 12] := "NeuroPLC_Weights".w1[6060 + lo] * (1.0 - t_val) + "NeuroPLC_Weights".w1[6060 + hi] * t_val;
    v3[15, 12] := "NeuroPLC_Weights".w1[6480 + lo] * (1.0 - t_val) + "NeuroPLC_Weights".w1[6480 + hi] * t_val;

    // --- Input 13: binary search ---
    lo := 0; hi := 14;
    WHILE hi - lo > 1 DO
        mid := lo + (hi - lo) / 2;
        IF v0[13] > "NeuroPLC_Weights".w0[mid] THEN lo := mid; ELSE hi := mid; END_IF;
    END_WHILE;
    t_val := (v0[13] - "NeuroPLC_Weights".w0[lo]) / ("NeuroPLC_Weights".w0[hi] - "NeuroPLC_Weights".w0[lo] + 1.0E-10);
    v3[0, 13] := "NeuroPLC_Weights".w1[195 + lo] * (1.0 - t_val) + "NeuroPLC_Weights".w1[195 + hi] * t_val;
    v3[1, 13] := "NeuroPLC_Weights".w1[615 + lo] * (1.0 - t_val) + "NeuroPLC_Weights".w1[615 + hi] * t_val;
    v3[2, 13] := "NeuroPLC_Weights".w1[1035 + lo] * (1.0 - t_val) + "NeuroPLC_Weights".w1[1035 + hi] * t_val;
    v3[3, 13] := "NeuroPLC_Weights".w1[1455 + lo] * (1.0 - t_val) + "NeuroPLC_Weights".w1[1455 + hi] * t_val;
    v3[4, 13] := "NeuroPLC_Weights".w1[1875 + lo] * (1.0 - t_val) + "NeuroPLC_Weights".w1[1875 + hi] * t_val;
    v3[5, 13] := "NeuroPLC_Weights".w1[2295 + lo] * (1.0 - t_val) + "NeuroPLC_Weights".w1[2295 + hi] * t_val;
    v3[6, 13] := "NeuroPLC_Weights".w1[2715 + lo] * (1.0 - t_val) + "NeuroPLC_Weights".w1[2715 + hi] * t_val;
    v3[7, 13] := "NeuroPLC_Weights".w1[3135 + lo] * (1.0 - t_val) + "NeuroPLC_Weights".w1[3135 + hi] * t_val;
    v3[8, 13] := "NeuroPLC_Weights".w1[3555 + lo] * (1.0 - t_val) + "NeuroPLC_Weights".w1[3555 + hi] * t_val;
    v3[9, 13] := "NeuroPLC_Weights".w1[3975 + lo] * (1.0 - t_val) + "NeuroPLC_Weights".w1[3975 + hi] * t_val;
    v3[10, 13] := "NeuroPLC_Weights".w1[4395 + lo] * (1.0 - t_val) + "NeuroPLC_Weights".w1[4395 + hi] * t_val;
    v3[11, 13] := "NeuroPLC_Weights".w1[4815 + lo] * (1.0 - t_val) + "NeuroPLC_Weights".w1[4815 + hi] * t_val;
    v3[12, 13] := "NeuroPLC_Weights".w1[5235 + lo] * (1.0 - t_val) + "NeuroPLC_Weights".w1[5235 + hi] * t_val;
    v3[13, 13] := "NeuroPLC_Weights".w1[5655 + lo] * (1.0 - t_val) + "NeuroPLC_Weights".w1[5655 + hi] * t_val;
    v3[14, 13] := "NeuroPLC_Weights".w1[6075 + lo] * (1.0 - t_val) + "NeuroPLC_Weights".w1[6075 + hi] * t_val;
    v3[15, 13] := "NeuroPLC_Weights".w1[6495 + lo] * (1.0 - t_val) + "NeuroPLC_Weights".w1[6495 + hi] * t_val;

    // --- Input 14: binary search ---
    lo := 0; hi := 14;
    WHILE hi - lo > 1 DO
        mid := lo + (hi - lo) / 2;
        IF v0[14] > "NeuroPLC_Weights".w0[mid] THEN lo := mid; ELSE hi := mid; END_IF;
    END_WHILE;
    t_val := (v0[14] - "NeuroPLC_Weights".w0[lo]) / ("NeuroPLC_Weights".w0[hi] - "NeuroPLC_Weights".w0[lo] + 1.0E-10);
    v3[0, 14] := "NeuroPLC_Weights".w1[210 + lo] * (1.0 - t_val) + "NeuroPLC_Weights".w1[210 + hi] * t_val;
    v3[1, 14] := "NeuroPLC_Weights".w1[630 + lo] * (1.0 - t_val) + "NeuroPLC_Weights".w1[630 + hi] * t_val;
    v3[2, 14] := "NeuroPLC_Weights".w1[1050 + lo] * (1.0 - t_val) + "NeuroPLC_Weights".w1[1050 + hi] * t_val;
    v3[3, 14] := "NeuroPLC_Weights".w1[1470 + lo] * (1.0 - t_val) + "NeuroPLC_Weights".w1[1470 + hi] * t_val;
    v3[4, 14] := "NeuroPLC_Weights".w1[1890 + lo] * (1.0 - t_val) + "NeuroPLC_Weights".w1[1890 + hi] * t_val;
    v3[5, 14] := "NeuroPLC_Weights".w1[2310 + lo] * (1.0 - t_val) + "NeuroPLC_Weights".w1[2310 + hi] * t_val;
    v3[6, 14] := "NeuroPLC_Weights".w1[2730 + lo] * (1.0 - t_val) + "NeuroPLC_Weights".w1[2730 + hi] * t_val;
    v3[7, 14] := "NeuroPLC_Weights".w1[3150 + lo] * (1.0 - t_val) + "NeuroPLC_Weights".w1[3150 + hi] * t_val;
    v3[8, 14] := "NeuroPLC_Weights".w1[3570 + lo] * (1.0 - t_val) + "NeuroPLC_Weights".w1[3570 + hi] * t_val;
    v3[9, 14] := "NeuroPLC_Weights".w1[3990 + lo] * (1.0 - t_val) + "NeuroPLC_Weights".w1[3990 + hi] * t_val;
    v3[10, 14] := "NeuroPLC_Weights".w1[4410 + lo] * (1.0 - t_val) + "NeuroPLC_Weights".w1[4410 + hi] * t_val;
    v3[11, 14] := "NeuroPLC_Weights".w1[4830 + lo] * (1.0 - t_val) + "NeuroPLC_Weights".w1[4830 + hi] * t_val;
    v3[12, 14] := "NeuroPLC_Weights".w1[5250 + lo] * (1.0 - t_val) + "NeuroPLC_Weights".w1[5250 + hi] * t_val;
    v3[13, 14] := "NeuroPLC_Weights".w1[5670 + lo] * (1.0 - t_val) + "NeuroPLC_Weights".w1[5670 + hi] * t_val;
    v3[14, 14] := "NeuroPLC_Weights".w1[6090 + lo] * (1.0 - t_val) + "NeuroPLC_Weights".w1[6090 + hi] * t_val;
    v3[15, 14] := "NeuroPLC_Weights".w1[6510 + lo] * (1.0 - t_val) + "NeuroPLC_Weights".w1[6510 + hi] * t_val;

    // --- Input 15: binary search ---
    lo := 0; hi := 14;
    WHILE hi - lo > 1 DO
        mid := lo + (hi - lo) / 2;
        IF v0[15] > "NeuroPLC_Weights".w0[mid] THEN lo := mid; ELSE hi := mid; END_IF;
    END_WHILE;
    t_val := (v0[15] - "NeuroPLC_Weights".w0[lo]) / ("NeuroPLC_Weights".w0[hi] - "NeuroPLC_Weights".w0[lo] + 1.0E-10);
    v3[0, 15] := "NeuroPLC_Weights".w1[225 + lo] * (1.0 - t_val) + "NeuroPLC_Weights".w1[225 + hi] * t_val;
    v3[1, 15] := "NeuroPLC_Weights".w1[645 + lo] * (1.0 - t_val) + "NeuroPLC_Weights".w1[645 + hi] * t_val;
    v3[2, 15] := "NeuroPLC_Weights".w1[1065 + lo] * (1.0 - t_val) + "NeuroPLC_Weights".w1[1065 + hi] * t_val;
    v3[3, 15] := "NeuroPLC_Weights".w1[1485 + lo] * (1.0 - t_val) + "NeuroPLC_Weights".w1[1485 + hi] * t_val;
    v3[4, 15] := "NeuroPLC_Weights".w1[1905 + lo] * (1.0 - t_val) + "NeuroPLC_Weights".w1[1905 + hi] * t_val;
    v3[5, 15] := "NeuroPLC_Weights".w1[2325 + lo] * (1.0 - t_val) + "NeuroPLC_Weights".w1[2325 + hi] * t_val;
    v3[6, 15] := "NeuroPLC_Weights".w1[2745 + lo] * (1.0 - t_val) + "NeuroPLC_Weights".w1[2745 + hi] * t_val;
    v3[7, 15] := "NeuroPLC_Weights".w1[3165 + lo] * (1.0 - t_val) + "NeuroPLC_Weights".w1[3165 + hi] * t_val;
    v3[8, 15] := "NeuroPLC_Weights".w1[3585 + lo] * (1.0 - t_val) + "NeuroPLC_Weights".w1[3585 + hi] * t_val;
    v3[9, 15] := "NeuroPLC_Weights".w1[4005 + lo] * (1.0 - t_val) + "NeuroPLC_Weights".w1[4005 + hi] * t_val;
    v3[10, 15] := "NeuroPLC_Weights".w1[4425 + lo] * (1.0 - t_val) + "NeuroPLC_Weights".w1[4425 + hi] * t_val;
    v3[11, 15] := "NeuroPLC_Weights".w1[4845 + lo] * (1.0 - t_val) + "NeuroPLC_Weights".w1[4845 + hi] * t_val;
    v3[12, 15] := "NeuroPLC_Weights".w1[5265 + lo] * (1.0 - t_val) + "NeuroPLC_Weights".w1[5265 + hi] * t_val;
    v3[13, 15] := "NeuroPLC_Weights".w1[5685 + lo] * (1.0 - t_val) + "NeuroPLC_Weights".w1[5685 + hi] * t_val;
    v3[14, 15] := "NeuroPLC_Weights".w1[6105 + lo] * (1.0 - t_val) + "NeuroPLC_Weights".w1[6105 + hi] * t_val;
    v3[15, 15] := "NeuroPLC_Weights".w1[6525 + lo] * (1.0 - t_val) + "NeuroPLC_Weights".w1[6525 + hi] * t_val;

    // --- Input 16: binary search ---
    lo := 0; hi := 14;
    WHILE hi - lo > 1 DO
        mid := lo + (hi - lo) / 2;
        IF v0[16] > "NeuroPLC_Weights".w0[mid] THEN lo := mid; ELSE hi := mid; END_IF;
    END_WHILE;
    t_val := (v0[16] - "NeuroPLC_Weights".w0[lo]) / ("NeuroPLC_Weights".w0[hi] - "NeuroPLC_Weights".w0[lo] + 1.0E-10);
    v3[0, 16] := "NeuroPLC_Weights".w1[240 + lo] * (1.0 - t_val) + "NeuroPLC_Weights".w1[240 + hi] * t_val;
    v3[1, 16] := "NeuroPLC_Weights".w1[660 + lo] * (1.0 - t_val) + "NeuroPLC_Weights".w1[660 + hi] * t_val;
    v3[2, 16] := "NeuroPLC_Weights".w1[1080 + lo] * (1.0 - t_val) + "NeuroPLC_Weights".w1[1080 + hi] * t_val;
    v3[3, 16] := "NeuroPLC_Weights".w1[1500 + lo] * (1.0 - t_val) + "NeuroPLC_Weights".w1[1500 + hi] * t_val;
    v3[4, 16] := "NeuroPLC_Weights".w1[1920 + lo] * (1.0 - t_val) + "NeuroPLC_Weights".w1[1920 + hi] * t_val;
    v3[5, 16] := "NeuroPLC_Weights".w1[2340 + lo] * (1.0 - t_val) + "NeuroPLC_Weights".w1[2340 + hi] * t_val;
    v3[6, 16] := "NeuroPLC_Weights".w1[2760 + lo] * (1.0 - t_val) + "NeuroPLC_Weights".w1[2760 + hi] * t_val;
    v3[7, 16] := "NeuroPLC_Weights".w1[3180 + lo] * (1.0 - t_val) + "NeuroPLC_Weights".w1[3180 + hi] * t_val;
    v3[8, 16] := "NeuroPLC_Weights".w1[3600 + lo] * (1.0 - t_val) + "NeuroPLC_Weights".w1[3600 + hi] * t_val;
    v3[9, 16] := "NeuroPLC_Weights".w1[4020 + lo] * (1.0 - t_val) + "NeuroPLC_Weights".w1[4020 + hi] * t_val;
    v3[10, 16] := "NeuroPLC_Weights".w1[4440 + lo] * (1.0 - t_val) + "NeuroPLC_Weights".w1[4440 + hi] * t_val;
    v3[11, 16] := "NeuroPLC_Weights".w1[4860 + lo] * (1.0 - t_val) + "NeuroPLC_Weights".w1[4860 + hi] * t_val;
    v3[12, 16] := "NeuroPLC_Weights".w1[5280 + lo] * (1.0 - t_val) + "NeuroPLC_Weights".w1[5280 + hi] * t_val;
    v3[13, 16] := "NeuroPLC_Weights".w1[5700 + lo] * (1.0 - t_val) + "NeuroPLC_Weights".w1[5700 + hi] * t_val;
    v3[14, 16] := "NeuroPLC_Weights".w1[6120 + lo] * (1.0 - t_val) + "NeuroPLC_Weights".w1[6120 + hi] * t_val;
    v3[15, 16] := "NeuroPLC_Weights".w1[6540 + lo] * (1.0 - t_val) + "NeuroPLC_Weights".w1[6540 + hi] * t_val;

    // --- Input 17: binary search ---
    lo := 0; hi := 14;
    WHILE hi - lo > 1 DO
        mid := lo + (hi - lo) / 2;
        IF v0[17] > "NeuroPLC_Weights".w0[mid] THEN lo := mid; ELSE hi := mid; END_IF;
    END_WHILE;
    t_val := (v0[17] - "NeuroPLC_Weights".w0[lo]) / ("NeuroPLC_Weights".w0[hi] - "NeuroPLC_Weights".w0[lo] + 1.0E-10);
    v3[0, 17] := "NeuroPLC_Weights".w1[255 + lo] * (1.0 - t_val) + "NeuroPLC_Weights".w1[255 + hi] * t_val;
    v3[1, 17] := "NeuroPLC_Weights".w1[675 + lo] * (1.0 - t_val) + "NeuroPLC_Weights".w1[675 + hi] * t_val;
    v3[2, 17] := "NeuroPLC_Weights".w1[1095 + lo] * (1.0 - t_val) + "NeuroPLC_Weights".w1[1095 + hi] * t_val;
    v3[3, 17] := "NeuroPLC_Weights".w1[1515 + lo] * (1.0 - t_val) + "NeuroPLC_Weights".w1[1515 + hi] * t_val;
    v3[4, 17] := "NeuroPLC_Weights".w1[1935 + lo] * (1.0 - t_val) + "NeuroPLC_Weights".w1[1935 + hi] * t_val;
    v3[5, 17] := "NeuroPLC_Weights".w1[2355 + lo] * (1.0 - t_val) + "NeuroPLC_Weights".w1[2355 + hi] * t_val;
    v3[6, 17] := "NeuroPLC_Weights".w1[2775 + lo] * (1.0 - t_val) + "NeuroPLC_Weights".w1[2775 + hi] * t_val;
    v3[7, 17] := "NeuroPLC_Weights".w1[3195 + lo] * (1.0 - t_val) + "NeuroPLC_Weights".w1[3195 + hi] * t_val;
    v3[8, 17] := "NeuroPLC_Weights".w1[3615 + lo] * (1.0 - t_val) + "NeuroPLC_Weights".w1[3615 + hi] * t_val;
    v3[9, 17] := "NeuroPLC_Weights".w1[4035 + lo] * (1.0 - t_val) + "NeuroPLC_Weights".w1[4035 + hi] * t_val;
    v3[10, 17] := "NeuroPLC_Weights".w1[4455 + lo] * (1.0 - t_val) + "NeuroPLC_Weights".w1[4455 + hi] * t_val;
    v3[11, 17] := "NeuroPLC_Weights".w1[4875 + lo] * (1.0 - t_val) + "NeuroPLC_Weights".w1[4875 + hi] * t_val;
    v3[12, 17] := "NeuroPLC_Weights".w1[5295 + lo] * (1.0 - t_val) + "NeuroPLC_Weights".w1[5295 + hi] * t_val;
    v3[13, 17] := "NeuroPLC_Weights".w1[5715 + lo] * (1.0 - t_val) + "NeuroPLC_Weights".w1[5715 + hi] * t_val;
    v3[14, 17] := "NeuroPLC_Weights".w1[6135 + lo] * (1.0 - t_val) + "NeuroPLC_Weights".w1[6135 + hi] * t_val;
    v3[15, 17] := "NeuroPLC_Weights".w1[6555 + lo] * (1.0 - t_val) + "NeuroPLC_Weights".w1[6555 + hi] * t_val;

    // --- Input 18: binary search ---
    lo := 0; hi := 14;
    WHILE hi - lo > 1 DO
        mid := lo + (hi - lo) / 2;
        IF v0[18] > "NeuroPLC_Weights".w0[mid] THEN lo := mid; ELSE hi := mid; END_IF;
    END_WHILE;
    t_val := (v0[18] - "NeuroPLC_Weights".w0[lo]) / ("NeuroPLC_Weights".w0[hi] - "NeuroPLC_Weights".w0[lo] + 1.0E-10);
    v3[0, 18] := "NeuroPLC_Weights".w1[270 + lo] * (1.0 - t_val) + "NeuroPLC_Weights".w1[270 + hi] * t_val;
    v3[1, 18] := "NeuroPLC_Weights".w1[690 + lo] * (1.0 - t_val) + "NeuroPLC_Weights".w1[690 + hi] * t_val;
    v3[2, 18] := "NeuroPLC_Weights".w1[1110 + lo] * (1.0 - t_val) + "NeuroPLC_Weights".w1[1110 + hi] * t_val;
    v3[3, 18] := "NeuroPLC_Weights".w1[1530 + lo] * (1.0 - t_val) + "NeuroPLC_Weights".w1[1530 + hi] * t_val;
    v3[4, 18] := "NeuroPLC_Weights".w1[1950 + lo] * (1.0 - t_val) + "NeuroPLC_Weights".w1[1950 + hi] * t_val;
    v3[5, 18] := "NeuroPLC_Weights".w1[2370 + lo] * (1.0 - t_val) + "NeuroPLC_Weights".w1[2370 + hi] * t_val;
    v3[6, 18] := "NeuroPLC_Weights".w1[2790 + lo] * (1.0 - t_val) + "NeuroPLC_Weights".w1[2790 + hi] * t_val;
    v3[7, 18] := "NeuroPLC_Weights".w1[3210 + lo] * (1.0 - t_val) + "NeuroPLC_Weights".w1[3210 + hi] * t_val;
    v3[8, 18] := "NeuroPLC_Weights".w1[3630 + lo] * (1.0 - t_val) + "NeuroPLC_Weights".w1[3630 + hi] * t_val;
    v3[9, 18] := "NeuroPLC_Weights".w1[4050 + lo] * (1.0 - t_val) + "NeuroPLC_Weights".w1[4050 + hi] * t_val;
    v3[10, 18] := "NeuroPLC_Weights".w1[4470 + lo] * (1.0 - t_val) + "NeuroPLC_Weights".w1[4470 + hi] * t_val;
    v3[11, 18] := "NeuroPLC_Weights".w1[4890 + lo] * (1.0 - t_val) + "NeuroPLC_Weights".w1[4890 + hi] * t_val;
    v3[12, 18] := "NeuroPLC_Weights".w1[5310 + lo] * (1.0 - t_val) + "NeuroPLC_Weights".w1[5310 + hi] * t_val;
    v3[13, 18] := "NeuroPLC_Weights".w1[5730 + lo] * (1.0 - t_val) + "NeuroPLC_Weights".w1[5730 + hi] * t_val;
    v3[14, 18] := "NeuroPLC_Weights".w1[6150 + lo] * (1.0 - t_val) + "NeuroPLC_Weights".w1[6150 + hi] * t_val;
    v3[15, 18] := "NeuroPLC_Weights".w1[6570 + lo] * (1.0 - t_val) + "NeuroPLC_Weights".w1[6570 + hi] * t_val;

    // --- Input 19: binary search ---
    lo := 0; hi := 14;
    WHILE hi - lo > 1 DO
        mid := lo + (hi - lo) / 2;
        IF v0[19] > "NeuroPLC_Weights".w0[mid] THEN lo := mid; ELSE hi := mid; END_IF;
    END_WHILE;
    t_val := (v0[19] - "NeuroPLC_Weights".w0[lo]) / ("NeuroPLC_Weights".w0[hi] - "NeuroPLC_Weights".w0[lo] + 1.0E-10);
    v3[0, 19] := "NeuroPLC_Weights".w1[285 + lo] * (1.0 - t_val) + "NeuroPLC_Weights".w1[285 + hi] * t_val;
    v3[1, 19] := "NeuroPLC_Weights".w1[705 + lo] * (1.0 - t_val) + "NeuroPLC_Weights".w1[705 + hi] * t_val;
    v3[2, 19] := "NeuroPLC_Weights".w1[1125 + lo] * (1.0 - t_val) + "NeuroPLC_Weights".w1[1125 + hi] * t_val;
    v3[3, 19] := "NeuroPLC_Weights".w1[1545 + lo] * (1.0 - t_val) + "NeuroPLC_Weights".w1[1545 + hi] * t_val;
    v3[4, 19] := "NeuroPLC_Weights".w1[1965 + lo] * (1.0 - t_val) + "NeuroPLC_Weights".w1[1965 + hi] * t_val;
    v3[5, 19] := "NeuroPLC_Weights".w1[2385 + lo] * (1.0 - t_val) + "NeuroPLC_Weights".w1[2385 + hi] * t_val;
    v3[6, 19] := "NeuroPLC_Weights".w1[2805 + lo] * (1.0 - t_val) + "NeuroPLC_Weights".w1[2805 + hi] * t_val;
    v3[7, 19] := "NeuroPLC_Weights".w1[3225 + lo] * (1.0 - t_val) + "NeuroPLC_Weights".w1[3225 + hi] * t_val;
    v3[8, 19] := "NeuroPLC_Weights".w1[3645 + lo] * (1.0 - t_val) + "NeuroPLC_Weights".w1[3645 + hi] * t_val;
    v3[9, 19] := "NeuroPLC_Weights".w1[4065 + lo] * (1.0 - t_val) + "NeuroPLC_Weights".w1[4065 + hi] * t_val;
    v3[10, 19] := "NeuroPLC_Weights".w1[4485 + lo] * (1.0 - t_val) + "NeuroPLC_Weights".w1[4485 + hi] * t_val;
    v3[11, 19] := "NeuroPLC_Weights".w1[4905 + lo] * (1.0 - t_val) + "NeuroPLC_Weights".w1[4905 + hi] * t_val;
    v3[12, 19] := "NeuroPLC_Weights".w1[5325 + lo] * (1.0 - t_val) + "NeuroPLC_Weights".w1[5325 + hi] * t_val;
    v3[13, 19] := "NeuroPLC_Weights".w1[5745 + lo] * (1.0 - t_val) + "NeuroPLC_Weights".w1[5745 + hi] * t_val;
    v3[14, 19] := "NeuroPLC_Weights".w1[6165 + lo] * (1.0 - t_val) + "NeuroPLC_Weights".w1[6165 + hi] * t_val;
    v3[15, 19] := "NeuroPLC_Weights".w1[6585 + lo] * (1.0 - t_val) + "NeuroPLC_Weights".w1[6585 + hi] * t_val;

    // --- Input 20: binary search ---
    lo := 0; hi := 14;
    WHILE hi - lo > 1 DO
        mid := lo + (hi - lo) / 2;
        IF v0[20] > "NeuroPLC_Weights".w0[mid] THEN lo := mid; ELSE hi := mid; END_IF;
    END_WHILE;
    t_val := (v0[20] - "NeuroPLC_Weights".w0[lo]) / ("NeuroPLC_Weights".w0[hi] - "NeuroPLC_Weights".w0[lo] + 1.0E-10);
    v3[0, 20] := "NeuroPLC_Weights".w1[300 + lo] * (1.0 - t_val) + "NeuroPLC_Weights".w1[300 + hi] * t_val;
    v3[1, 20] := "NeuroPLC_Weights".w1[720 + lo] * (1.0 - t_val) + "NeuroPLC_Weights".w1[720 + hi] * t_val;
    v3[2, 20] := "NeuroPLC_Weights".w1[1140 + lo] * (1.0 - t_val) + "NeuroPLC_Weights".w1[1140 + hi] * t_val;
    v3[3, 20] := "NeuroPLC_Weights".w1[1560 + lo] * (1.0 - t_val) + "NeuroPLC_Weights".w1[1560 + hi] * t_val;
    v3[4, 20] := "NeuroPLC_Weights".w1[1980 + lo] * (1.0 - t_val) + "NeuroPLC_Weights".w1[1980 + hi] * t_val;
    v3[5, 20] := "NeuroPLC_Weights".w1[2400 + lo] * (1.0 - t_val) + "NeuroPLC_Weights".w1[2400 + hi] * t_val;
    v3[6, 20] := "NeuroPLC_Weights".w1[2820 + lo] * (1.0 - t_val) + "NeuroPLC_Weights".w1[2820 + hi] * t_val;
    v3[7, 20] := "NeuroPLC_Weights".w1[3240 + lo] * (1.0 - t_val) + "NeuroPLC_Weights".w1[3240 + hi] * t_val;
    v3[8, 20] := "NeuroPLC_Weights".w1[3660 + lo] * (1.0 - t_val) + "NeuroPLC_Weights".w1[3660 + hi] * t_val;
    v3[9, 20] := "NeuroPLC_Weights".w1[4080 + lo] * (1.0 - t_val) + "NeuroPLC_Weights".w1[4080 + hi] * t_val;
    v3[10, 20] := "NeuroPLC_Weights".w1[4500 + lo] * (1.0 - t_val) + "NeuroPLC_Weights".w1[4500 + hi] * t_val;
    v3[11, 20] := "NeuroPLC_Weights".w1[4920 + lo] * (1.0 - t_val) + "NeuroPLC_Weights".w1[4920 + hi] * t_val;
    v3[12, 20] := "NeuroPLC_Weights".w1[5340 + lo] * (1.0 - t_val) + "NeuroPLC_Weights".w1[5340 + hi] * t_val;
    v3[13, 20] := "NeuroPLC_Weights".w1[5760 + lo] * (1.0 - t_val) + "NeuroPLC_Weights".w1[5760 + hi] * t_val;
    v3[14, 20] := "NeuroPLC_Weights".w1[6180 + lo] * (1.0 - t_val) + "NeuroPLC_Weights".w1[6180 + hi] * t_val;
    v3[15, 20] := "NeuroPLC_Weights".w1[6600 + lo] * (1.0 - t_val) + "NeuroPLC_Weights".w1[6600 + hi] * t_val;

    // --- Input 21: binary search ---
    lo := 0; hi := 14;
    WHILE hi - lo > 1 DO
        mid := lo + (hi - lo) / 2;
        IF v0[21] > "NeuroPLC_Weights".w0[mid] THEN lo := mid; ELSE hi := mid; END_IF;
    END_WHILE;
    t_val := (v0[21] - "NeuroPLC_Weights".w0[lo]) / ("NeuroPLC_Weights".w0[hi] - "NeuroPLC_Weights".w0[lo] + 1.0E-10);
    v3[0, 21] := "NeuroPLC_Weights".w1[315 + lo] * (1.0 - t_val) + "NeuroPLC_Weights".w1[315 + hi] * t_val;
    v3[1, 21] := "NeuroPLC_Weights".w1[735 + lo] * (1.0 - t_val) + "NeuroPLC_Weights".w1[735 + hi] * t_val;
    v3[2, 21] := "NeuroPLC_Weights".w1[1155 + lo] * (1.0 - t_val) + "NeuroPLC_Weights".w1[1155 + hi] * t_val;
    v3[3, 21] := "NeuroPLC_Weights".w1[1575 + lo] * (1.0 - t_val) + "NeuroPLC_Weights".w1[1575 + hi] * t_val;
    v3[4, 21] := "NeuroPLC_Weights".w1[1995 + lo] * (1.0 - t_val) + "NeuroPLC_Weights".w1[1995 + hi] * t_val;
    v3[5, 21] := "NeuroPLC_Weights".w1[2415 + lo] * (1.0 - t_val) + "NeuroPLC_Weights".w1[2415 + hi] * t_val;
    v3[6, 21] := "NeuroPLC_Weights".w1[2835 + lo] * (1.0 - t_val) + "NeuroPLC_Weights".w1[2835 + hi] * t_val;
    v3[7, 21] := "NeuroPLC_Weights".w1[3255 + lo] * (1.0 - t_val) + "NeuroPLC_Weights".w1[3255 + hi] * t_val;
    v3[8, 21] := "NeuroPLC_Weights".w1[3675 + lo] * (1.0 - t_val) + "NeuroPLC_Weights".w1[3675 + hi] * t_val;
    v3[9, 21] := "NeuroPLC_Weights".w1[4095 + lo] * (1.0 - t_val) + "NeuroPLC_Weights".w1[4095 + hi] * t_val;
    v3[10, 21] := "NeuroPLC_Weights".w1[4515 + lo] * (1.0 - t_val) + "NeuroPLC_Weights".w1[4515 + hi] * t_val;
    v3[11, 21] := "NeuroPLC_Weights".w1[4935 + lo] * (1.0 - t_val) + "NeuroPLC_Weights".w1[4935 + hi] * t_val;
    v3[12, 21] := "NeuroPLC_Weights".w1[5355 + lo] * (1.0 - t_val) + "NeuroPLC_Weights".w1[5355 + hi] * t_val;
    v3[13, 21] := "NeuroPLC_Weights".w1[5775 + lo] * (1.0 - t_val) + "NeuroPLC_Weights".w1[5775 + hi] * t_val;
    v3[14, 21] := "NeuroPLC_Weights".w1[6195 + lo] * (1.0 - t_val) + "NeuroPLC_Weights".w1[6195 + hi] * t_val;
    v3[15, 21] := "NeuroPLC_Weights".w1[6615 + lo] * (1.0 - t_val) + "NeuroPLC_Weights".w1[6615 + hi] * t_val;

    // --- Input 22: binary search ---
    lo := 0; hi := 14;
    WHILE hi - lo > 1 DO
        mid := lo + (hi - lo) / 2;
        IF v0[22] > "NeuroPLC_Weights".w0[mid] THEN lo := mid; ELSE hi := mid; END_IF;
    END_WHILE;
    t_val := (v0[22] - "NeuroPLC_Weights".w0[lo]) / ("NeuroPLC_Weights".w0[hi] - "NeuroPLC_Weights".w0[lo] + 1.0E-10);
    v3[0, 22] := "NeuroPLC_Weights".w1[330 + lo] * (1.0 - t_val) + "NeuroPLC_Weights".w1[330 + hi] * t_val;
    v3[1, 22] := "NeuroPLC_Weights".w1[750 + lo] * (1.0 - t_val) + "NeuroPLC_Weights".w1[750 + hi] * t_val;
    v3[2, 22] := "NeuroPLC_Weights".w1[1170 + lo] * (1.0 - t_val) + "NeuroPLC_Weights".w1[1170 + hi] * t_val;
    v3[3, 22] := "NeuroPLC_Weights".w1[1590 + lo] * (1.0 - t_val) + "NeuroPLC_Weights".w1[1590 + hi] * t_val;
    v3[4, 22] := "NeuroPLC_Weights".w1[2010 + lo] * (1.0 - t_val) + "NeuroPLC_Weights".w1[2010 + hi] * t_val;
    v3[5, 22] := "NeuroPLC_Weights".w1[2430 + lo] * (1.0 - t_val) + "NeuroPLC_Weights".w1[2430 + hi] * t_val;
    v3[6, 22] := "NeuroPLC_Weights".w1[2850 + lo] * (1.0 - t_val) + "NeuroPLC_Weights".w1[2850 + hi] * t_val;
    v3[7, 22] := "NeuroPLC_Weights".w1[3270 + lo] * (1.0 - t_val) + "NeuroPLC_Weights".w1[3270 + hi] * t_val;
    v3[8, 22] := "NeuroPLC_Weights".w1[3690 + lo] * (1.0 - t_val) + "NeuroPLC_Weights".w1[3690 + hi] * t_val;
    v3[9, 22] := "NeuroPLC_Weights".w1[4110 + lo] * (1.0 - t_val) + "NeuroPLC_Weights".w1[4110 + hi] * t_val;
    v3[10, 22] := "NeuroPLC_Weights".w1[4530 + lo] * (1.0 - t_val) + "NeuroPLC_Weights".w1[4530 + hi] * t_val;
    v3[11, 22] := "NeuroPLC_Weights".w1[4950 + lo] * (1.0 - t_val) + "NeuroPLC_Weights".w1[4950 + hi] * t_val;
    v3[12, 22] := "NeuroPLC_Weights".w1[5370 + lo] * (1.0 - t_val) + "NeuroPLC_Weights".w1[5370 + hi] * t_val;
    v3[13, 22] := "NeuroPLC_Weights".w1[5790 + lo] * (1.0 - t_val) + "NeuroPLC_Weights".w1[5790 + hi] * t_val;
    v3[14, 22] := "NeuroPLC_Weights".w1[6210 + lo] * (1.0 - t_val) + "NeuroPLC_Weights".w1[6210 + hi] * t_val;
    v3[15, 22] := "NeuroPLC_Weights".w1[6630 + lo] * (1.0 - t_val) + "NeuroPLC_Weights".w1[6630 + hi] * t_val;

    // --- Input 23: binary search ---
    lo := 0; hi := 14;
    WHILE hi - lo > 1 DO
        mid := lo + (hi - lo) / 2;
        IF v0[23] > "NeuroPLC_Weights".w0[mid] THEN lo := mid; ELSE hi := mid; END_IF;
    END_WHILE;
    t_val := (v0[23] - "NeuroPLC_Weights".w0[lo]) / ("NeuroPLC_Weights".w0[hi] - "NeuroPLC_Weights".w0[lo] + 1.0E-10);
    v3[0, 23] := "NeuroPLC_Weights".w1[345 + lo] * (1.0 - t_val) + "NeuroPLC_Weights".w1[345 + hi] * t_val;
    v3[1, 23] := "NeuroPLC_Weights".w1[765 + lo] * (1.0 - t_val) + "NeuroPLC_Weights".w1[765 + hi] * t_val;
    v3[2, 23] := "NeuroPLC_Weights".w1[1185 + lo] * (1.0 - t_val) + "NeuroPLC_Weights".w1[1185 + hi] * t_val;
    v3[3, 23] := "NeuroPLC_Weights".w1[1605 + lo] * (1.0 - t_val) + "NeuroPLC_Weights".w1[1605 + hi] * t_val;
    v3[4, 23] := "NeuroPLC_Weights".w1[2025 + lo] * (1.0 - t_val) + "NeuroPLC_Weights".w1[2025 + hi] * t_val;
    v3[5, 23] := "NeuroPLC_Weights".w1[2445 + lo] * (1.0 - t_val) + "NeuroPLC_Weights".w1[2445 + hi] * t_val;
    v3[6, 23] := "NeuroPLC_Weights".w1[2865 + lo] * (1.0 - t_val) + "NeuroPLC_Weights".w1[2865 + hi] * t_val;
    v3[7, 23] := "NeuroPLC_Weights".w1[3285 + lo] * (1.0 - t_val) + "NeuroPLC_Weights".w1[3285 + hi] * t_val;
    v3[8, 23] := "NeuroPLC_Weights".w1[3705 + lo] * (1.0 - t_val) + "NeuroPLC_Weights".w1[3705 + hi] * t_val;
    v3[9, 23] := "NeuroPLC_Weights".w1[4125 + lo] * (1.0 - t_val) + "NeuroPLC_Weights".w1[4125 + hi] * t_val;
    v3[10, 23] := "NeuroPLC_Weights".w1[4545 + lo] * (1.0 - t_val) + "NeuroPLC_Weights".w1[4545 + hi] * t_val;
    v3[11, 23] := "NeuroPLC_Weights".w1[4965 + lo] * (1.0 - t_val) + "NeuroPLC_Weights".w1[4965 + hi] * t_val;
    v3[12, 23] := "NeuroPLC_Weights".w1[5385 + lo] * (1.0 - t_val) + "NeuroPLC_Weights".w1[5385 + hi] * t_val;
    v3[13, 23] := "NeuroPLC_Weights".w1[5805 + lo] * (1.0 - t_val) + "NeuroPLC_Weights".w1[5805 + hi] * t_val;
    v3[14, 23] := "NeuroPLC_Weights".w1[6225 + lo] * (1.0 - t_val) + "NeuroPLC_Weights".w1[6225 + hi] * t_val;
    v3[15, 23] := "NeuroPLC_Weights".w1[6645 + lo] * (1.0 - t_val) + "NeuroPLC_Weights".w1[6645 + hi] * t_val;

    // --- Input 24: binary search ---
    lo := 0; hi := 14;
    WHILE hi - lo > 1 DO
        mid := lo + (hi - lo) / 2;
        IF v0[24] > "NeuroPLC_Weights".w0[mid] THEN lo := mid; ELSE hi := mid; END_IF;
    END_WHILE;
    t_val := (v0[24] - "NeuroPLC_Weights".w0[lo]) / ("NeuroPLC_Weights".w0[hi] - "NeuroPLC_Weights".w0[lo] + 1.0E-10);
    v3[0, 24] := "NeuroPLC_Weights".w1[360 + lo] * (1.0 - t_val) + "NeuroPLC_Weights".w1[360 + hi] * t_val;
    v3[1, 24] := "NeuroPLC_Weights".w1[780 + lo] * (1.0 - t_val) + "NeuroPLC_Weights".w1[780 + hi] * t_val;
    v3[2, 24] := "NeuroPLC_Weights".w1[1200 + lo] * (1.0 - t_val) + "NeuroPLC_Weights".w1[1200 + hi] * t_val;
    v3[3, 24] := "NeuroPLC_Weights".w1[1620 + lo] * (1.0 - t_val) + "NeuroPLC_Weights".w1[1620 + hi] * t_val;
    v3[4, 24] := "NeuroPLC_Weights".w1[2040 + lo] * (1.0 - t_val) + "NeuroPLC_Weights".w1[2040 + hi] * t_val;
    v3[5, 24] := "NeuroPLC_Weights".w1[2460 + lo] * (1.0 - t_val) + "NeuroPLC_Weights".w1[2460 + hi] * t_val;
    v3[6, 24] := "NeuroPLC_Weights".w1[2880 + lo] * (1.0 - t_val) + "NeuroPLC_Weights".w1[2880 + hi] * t_val;
    v3[7, 24] := "NeuroPLC_Weights".w1[3300 + lo] * (1.0 - t_val) + "NeuroPLC_Weights".w1[3300 + hi] * t_val;
    v3[8, 24] := "NeuroPLC_Weights".w1[3720 + lo] * (1.0 - t_val) + "NeuroPLC_Weights".w1[3720 + hi] * t_val;
    v3[9, 24] := "NeuroPLC_Weights".w1[4140 + lo] * (1.0 - t_val) + "NeuroPLC_Weights".w1[4140 + hi] * t_val;
    v3[10, 24] := "NeuroPLC_Weights".w1[4560 + lo] * (1.0 - t_val) + "NeuroPLC_Weights".w1[4560 + hi] * t_val;
    v3[11, 24] := "NeuroPLC_Weights".w1[4980 + lo] * (1.0 - t_val) + "NeuroPLC_Weights".w1[4980 + hi] * t_val;
    v3[12, 24] := "NeuroPLC_Weights".w1[5400 + lo] * (1.0 - t_val) + "NeuroPLC_Weights".w1[5400 + hi] * t_val;
    v3[13, 24] := "NeuroPLC_Weights".w1[5820 + lo] * (1.0 - t_val) + "NeuroPLC_Weights".w1[5820 + hi] * t_val;
    v3[14, 24] := "NeuroPLC_Weights".w1[6240 + lo] * (1.0 - t_val) + "NeuroPLC_Weights".w1[6240 + hi] * t_val;
    v3[15, 24] := "NeuroPLC_Weights".w1[6660 + lo] * (1.0 - t_val) + "NeuroPLC_Weights".w1[6660 + hi] * t_val;

    // --- Input 25: binary search ---
    lo := 0; hi := 14;
    WHILE hi - lo > 1 DO
        mid := lo + (hi - lo) / 2;
        IF v0[25] > "NeuroPLC_Weights".w0[mid] THEN lo := mid; ELSE hi := mid; END_IF;
    END_WHILE;
    t_val := (v0[25] - "NeuroPLC_Weights".w0[lo]) / ("NeuroPLC_Weights".w0[hi] - "NeuroPLC_Weights".w0[lo] + 1.0E-10);
    v3[0, 25] := "NeuroPLC_Weights".w1[375 + lo] * (1.0 - t_val) + "NeuroPLC_Weights".w1[375 + hi] * t_val;
    v3[1, 25] := "NeuroPLC_Weights".w1[795 + lo] * (1.0 - t_val) + "NeuroPLC_Weights".w1[795 + hi] * t_val;
    v3[2, 25] := "NeuroPLC_Weights".w1[1215 + lo] * (1.0 - t_val) + "NeuroPLC_Weights".w1[1215 + hi] * t_val;
    v3[3, 25] := "NeuroPLC_Weights".w1[1635 + lo] * (1.0 - t_val) + "NeuroPLC_Weights".w1[1635 + hi] * t_val;
    v3[4, 25] := "NeuroPLC_Weights".w1[2055 + lo] * (1.0 - t_val) + "NeuroPLC_Weights".w1[2055 + hi] * t_val;
    v3[5, 25] := "NeuroPLC_Weights".w1[2475 + lo] * (1.0 - t_val) + "NeuroPLC_Weights".w1[2475 + hi] * t_val;
    v3[6, 25] := "NeuroPLC_Weights".w1[2895 + lo] * (1.0 - t_val) + "NeuroPLC_Weights".w1[2895 + hi] * t_val;
    v3[7, 25] := "NeuroPLC_Weights".w1[3315 + lo] * (1.0 - t_val) + "NeuroPLC_Weights".w1[3315 + hi] * t_val;
    v3[8, 25] := "NeuroPLC_Weights".w1[3735 + lo] * (1.0 - t_val) + "NeuroPLC_Weights".w1[3735 + hi] * t_val;
    v3[9, 25] := "NeuroPLC_Weights".w1[4155 + lo] * (1.0 - t_val) + "NeuroPLC_Weights".w1[4155 + hi] * t_val;
    v3[10, 25] := "NeuroPLC_Weights".w1[4575 + lo] * (1.0 - t_val) + "NeuroPLC_Weights".w1[4575 + hi] * t_val;
    v3[11, 25] := "NeuroPLC_Weights".w1[4995 + lo] * (1.0 - t_val) + "NeuroPLC_Weights".w1[4995 + hi] * t_val;
    v3[12, 25] := "NeuroPLC_Weights".w1[5415 + lo] * (1.0 - t_val) + "NeuroPLC_Weights".w1[5415 + hi] * t_val;
    v3[13, 25] := "NeuroPLC_Weights".w1[5835 + lo] * (1.0 - t_val) + "NeuroPLC_Weights".w1[5835 + hi] * t_val;
    v3[14, 25] := "NeuroPLC_Weights".w1[6255 + lo] * (1.0 - t_val) + "NeuroPLC_Weights".w1[6255 + hi] * t_val;
    v3[15, 25] := "NeuroPLC_Weights".w1[6675 + lo] * (1.0 - t_val) + "NeuroPLC_Weights".w1[6675 + hi] * t_val;

    // --- Input 26: binary search ---
    lo := 0; hi := 14;
    WHILE hi - lo > 1 DO
        mid := lo + (hi - lo) / 2;
        IF v0[26] > "NeuroPLC_Weights".w0[mid] THEN lo := mid; ELSE hi := mid; END_IF;
    END_WHILE;
    t_val := (v0[26] - "NeuroPLC_Weights".w0[lo]) / ("NeuroPLC_Weights".w0[hi] - "NeuroPLC_Weights".w0[lo] + 1.0E-10);
    v3[0, 26] := "NeuroPLC_Weights".w1[390 + lo] * (1.0 - t_val) + "NeuroPLC_Weights".w1[390 + hi] * t_val;
    v3[1, 26] := "NeuroPLC_Weights".w1[810 + lo] * (1.0 - t_val) + "NeuroPLC_Weights".w1[810 + hi] * t_val;
    v3[2, 26] := "NeuroPLC_Weights".w1[1230 + lo] * (1.0 - t_val) + "NeuroPLC_Weights".w1[1230 + hi] * t_val;
    v3[3, 26] := "NeuroPLC_Weights".w1[1650 + lo] * (1.0 - t_val) + "NeuroPLC_Weights".w1[1650 + hi] * t_val;
    v3[4, 26] := "NeuroPLC_Weights".w1[2070 + lo] * (1.0 - t_val) + "NeuroPLC_Weights".w1[2070 + hi] * t_val;
    v3[5, 26] := "NeuroPLC_Weights".w1[2490 + lo] * (1.0 - t_val) + "NeuroPLC_Weights".w1[2490 + hi] * t_val;
    v3[6, 26] := "NeuroPLC_Weights".w1[2910 + lo] * (1.0 - t_val) + "NeuroPLC_Weights".w1[2910 + hi] * t_val;
    v3[7, 26] := "NeuroPLC_Weights".w1[3330 + lo] * (1.0 - t_val) + "NeuroPLC_Weights".w1[3330 + hi] * t_val;
    v3[8, 26] := "NeuroPLC_Weights".w1[3750 + lo] * (1.0 - t_val) + "NeuroPLC_Weights".w1[3750 + hi] * t_val;
    v3[9, 26] := "NeuroPLC_Weights".w1[4170 + lo] * (1.0 - t_val) + "NeuroPLC_Weights".w1[4170 + hi] * t_val;
    v3[10, 26] := "NeuroPLC_Weights".w1[4590 + lo] * (1.0 - t_val) + "NeuroPLC_Weights".w1[4590 + hi] * t_val;
    v3[11, 26] := "NeuroPLC_Weights".w1[5010 + lo] * (1.0 - t_val) + "NeuroPLC_Weights".w1[5010 + hi] * t_val;
    v3[12, 26] := "NeuroPLC_Weights".w1[5430 + lo] * (1.0 - t_val) + "NeuroPLC_Weights".w1[5430 + hi] * t_val;
    v3[13, 26] := "NeuroPLC_Weights".w1[5850 + lo] * (1.0 - t_val) + "NeuroPLC_Weights".w1[5850 + hi] * t_val;
    v3[14, 26] := "NeuroPLC_Weights".w1[6270 + lo] * (1.0 - t_val) + "NeuroPLC_Weights".w1[6270 + hi] * t_val;
    v3[15, 26] := "NeuroPLC_Weights".w1[6690 + lo] * (1.0 - t_val) + "NeuroPLC_Weights".w1[6690 + hi] * t_val;

    // --- Input 27: binary search ---
    lo := 0; hi := 14;
    WHILE hi - lo > 1 DO
        mid := lo + (hi - lo) / 2;
        IF v0[27] > "NeuroPLC_Weights".w0[mid] THEN lo := mid; ELSE hi := mid; END_IF;
    END_WHILE;
    t_val := (v0[27] - "NeuroPLC_Weights".w0[lo]) / ("NeuroPLC_Weights".w0[hi] - "NeuroPLC_Weights".w0[lo] + 1.0E-10);
    v3[0, 27] := "NeuroPLC_Weights".w1[405 + lo] * (1.0 - t_val) + "NeuroPLC_Weights".w1[405 + hi] * t_val;
    v3[1, 27] := "NeuroPLC_Weights".w1[825 + lo] * (1.0 - t_val) + "NeuroPLC_Weights".w1[825 + hi] * t_val;
    v3[2, 27] := "NeuroPLC_Weights".w1[1245 + lo] * (1.0 - t_val) + "NeuroPLC_Weights".w1[1245 + hi] * t_val;
    v3[3, 27] := "NeuroPLC_Weights".w1[1665 + lo] * (1.0 - t_val) + "NeuroPLC_Weights".w1[1665 + hi] * t_val;
    v3[4, 27] := "NeuroPLC_Weights".w1[2085 + lo] * (1.0 - t_val) + "NeuroPLC_Weights".w1[2085 + hi] * t_val;
    v3[5, 27] := "NeuroPLC_Weights".w1[2505 + lo] * (1.0 - t_val) + "NeuroPLC_Weights".w1[2505 + hi] * t_val;
    v3[6, 27] := "NeuroPLC_Weights".w1[2925 + lo] * (1.0 - t_val) + "NeuroPLC_Weights".w1[2925 + hi] * t_val;
    v3[7, 27] := "NeuroPLC_Weights".w1[3345 + lo] * (1.0 - t_val) + "NeuroPLC_Weights".w1[3345 + hi] * t_val;
    v3[8, 27] := "NeuroPLC_Weights".w1[3765 + lo] * (1.0 - t_val) + "NeuroPLC_Weights".w1[3765 + hi] * t_val;
    v3[9, 27] := "NeuroPLC_Weights".w1[4185 + lo] * (1.0 - t_val) + "NeuroPLC_Weights".w1[4185 + hi] * t_val;
    v3[10, 27] := "NeuroPLC_Weights".w1[4605 + lo] * (1.0 - t_val) + "NeuroPLC_Weights".w1[4605 + hi] * t_val;
    v3[11, 27] := "NeuroPLC_Weights".w1[5025 + lo] * (1.0 - t_val) + "NeuroPLC_Weights".w1[5025 + hi] * t_val;
    v3[12, 27] := "NeuroPLC_Weights".w1[5445 + lo] * (1.0 - t_val) + "NeuroPLC_Weights".w1[5445 + hi] * t_val;
    v3[13, 27] := "NeuroPLC_Weights".w1[5865 + lo] * (1.0 - t_val) + "NeuroPLC_Weights".w1[5865 + hi] * t_val;
    v3[14, 27] := "NeuroPLC_Weights".w1[6285 + lo] * (1.0 - t_val) + "NeuroPLC_Weights".w1[6285 + hi] * t_val;
    v3[15, 27] := "NeuroPLC_Weights".w1[6705 + lo] * (1.0 - t_val) + "NeuroPLC_Weights".w1[6705 + hi] * t_val;


    // ---- l0_base: MatMul(28→16) ----
    // W = "NeuroPLC_Weights".w2[:448],   b = w2[448:]
    v2[0] := "NeuroPLC_Weights".w2[448 + 0];
    FOR i := 0 TO 27 DO
        v2[0] := v2[0] + "NeuroPLC_Weights".w2[0 + i] * v1[i];
    END_FOR;
    v2[1] := "NeuroPLC_Weights".w2[448 + 1];
    FOR i := 0 TO 27 DO
        v2[1] := v2[1] + "NeuroPLC_Weights".w2[28 + i] * v1[i];
    END_FOR;
    v2[2] := "NeuroPLC_Weights".w2[448 + 2];
    FOR i := 0 TO 27 DO
        v2[2] := v2[2] + "NeuroPLC_Weights".w2[56 + i] * v1[i];
    END_FOR;
    v2[3] := "NeuroPLC_Weights".w2[448 + 3];
    FOR i := 0 TO 27 DO
        v2[3] := v2[3] + "NeuroPLC_Weights".w2[84 + i] * v1[i];
    END_FOR;
    v2[4] := "NeuroPLC_Weights".w2[448 + 4];
    FOR i := 0 TO 27 DO
        v2[4] := v2[4] + "NeuroPLC_Weights".w2[112 + i] * v1[i];
    END_FOR;
    v2[5] := "NeuroPLC_Weights".w2[448 + 5];
    FOR i := 0 TO 27 DO
        v2[5] := v2[5] + "NeuroPLC_Weights".w2[140 + i] * v1[i];
    END_FOR;
    v2[6] := "NeuroPLC_Weights".w2[448 + 6];
    FOR i := 0 TO 27 DO
        v2[6] := v2[6] + "NeuroPLC_Weights".w2[168 + i] * v1[i];
    END_FOR;
    v2[7] := "NeuroPLC_Weights".w2[448 + 7];
    FOR i := 0 TO 27 DO
        v2[7] := v2[7] + "NeuroPLC_Weights".w2[196 + i] * v1[i];
    END_FOR;
    v2[8] := "NeuroPLC_Weights".w2[448 + 8];
    FOR i := 0 TO 27 DO
        v2[8] := v2[8] + "NeuroPLC_Weights".w2[224 + i] * v1[i];
    END_FOR;
    v2[9] := "NeuroPLC_Weights".w2[448 + 9];
    FOR i := 0 TO 27 DO
        v2[9] := v2[9] + "NeuroPLC_Weights".w2[252 + i] * v1[i];
    END_FOR;
    v2[10] := "NeuroPLC_Weights".w2[448 + 10];
    FOR i := 0 TO 27 DO
        v2[10] := v2[10] + "NeuroPLC_Weights".w2[280 + i] * v1[i];
    END_FOR;
    v2[11] := "NeuroPLC_Weights".w2[448 + 11];
    FOR i := 0 TO 27 DO
        v2[11] := v2[11] + "NeuroPLC_Weights".w2[308 + i] * v1[i];
    END_FOR;
    v2[12] := "NeuroPLC_Weights".w2[448 + 12];
    FOR i := 0 TO 27 DO
        v2[12] := v2[12] + "NeuroPLC_Weights".w2[336 + i] * v1[i];
    END_FOR;
    v2[13] := "NeuroPLC_Weights".w2[448 + 13];
    FOR i := 0 TO 27 DO
        v2[13] := v2[13] + "NeuroPLC_Weights".w2[364 + i] * v1[i];
    END_FOR;
    v2[14] := "NeuroPLC_Weights".w2[448 + 14];
    FOR i := 0 TO 27 DO
        v2[14] := v2[14] + "NeuroPLC_Weights".w2[392 + i] * v1[i];
    END_FOR;
    v2[15] := "NeuroPLC_Weights".w2[448 + 15];
    FOR i := 0 TO 27 DO
        v2[15] := v2[15] + "NeuroPLC_Weights".w2[420 + i] * v1[i];
    END_FOR;

    // ---- l0_merge: Add (KAN merge) ----
    v4[0] := v2[0] + v3[0, 0] + v3[0, 1] + v3[0, 2] + v3[0, 3] + v3[0, 4] + v3[0, 5] + v3[0, 6] + v3[0, 7] + v3[0, 8] + v3[0, 9] + v3[0, 10] + v3[0, 11] + v3[0, 12] + v3[0, 13] + v3[0, 14] + v3[0, 15] + v3[0, 16] + v3[0, 17] + v3[0, 18] + v3[0, 19] + v3[0, 20] + v3[0, 21] + v3[0, 22] + v3[0, 23] + v3[0, 24] + v3[0, 25] + v3[0, 26] + v3[0, 27];
    v4[1] := v2[1] + v3[1, 0] + v3[1, 1] + v3[1, 2] + v3[1, 3] + v3[1, 4] + v3[1, 5] + v3[1, 6] + v3[1, 7] + v3[1, 8] + v3[1, 9] + v3[1, 10] + v3[1, 11] + v3[1, 12] + v3[1, 13] + v3[1, 14] + v3[1, 15] + v3[1, 16] + v3[1, 17] + v3[1, 18] + v3[1, 19] + v3[1, 20] + v3[1, 21] + v3[1, 22] + v3[1, 23] + v3[1, 24] + v3[1, 25] + v3[1, 26] + v3[1, 27];
    v4[2] := v2[2] + v3[2, 0] + v3[2, 1] + v3[2, 2] + v3[2, 3] + v3[2, 4] + v3[2, 5] + v3[2, 6] + v3[2, 7] + v3[2, 8] + v3[2, 9] + v3[2, 10] + v3[2, 11] + v3[2, 12] + v3[2, 13] + v3[2, 14] + v3[2, 15] + v3[2, 16] + v3[2, 17] + v3[2, 18] + v3[2, 19] + v3[2, 20] + v3[2, 21] + v3[2, 22] + v3[2, 23] + v3[2, 24] + v3[2, 25] + v3[2, 26] + v3[2, 27];
    v4[3] := v2[3] + v3[3, 0] + v3[3, 1] + v3[3, 2] + v3[3, 3] + v3[3, 4] + v3[3, 5] + v3[3, 6] + v3[3, 7] + v3[3, 8] + v3[3, 9] + v3[3, 10] + v3[3, 11] + v3[3, 12] + v3[3, 13] + v3[3, 14] + v3[3, 15] + v3[3, 16] + v3[3, 17] + v3[3, 18] + v3[3, 19] + v3[3, 20] + v3[3, 21] + v3[3, 22] + v3[3, 23] + v3[3, 24] + v3[3, 25] + v3[3, 26] + v3[3, 27];
    v4[4] := v2[4] + v3[4, 0] + v3[4, 1] + v3[4, 2] + v3[4, 3] + v3[4, 4] + v3[4, 5] + v3[4, 6] + v3[4, 7] + v3[4, 8] + v3[4, 9] + v3[4, 10] + v3[4, 11] + v3[4, 12] + v3[4, 13] + v3[4, 14] + v3[4, 15] + v3[4, 16] + v3[4, 17] + v3[4, 18] + v3[4, 19] + v3[4, 20] + v3[4, 21] + v3[4, 22] + v3[4, 23] + v3[4, 24] + v3[4, 25] + v3[4, 26] + v3[4, 27];
    v4[5] := v2[5] + v3[5, 0] + v3[5, 1] + v3[5, 2] + v3[5, 3] + v3[5, 4] + v3[5, 5] + v3[5, 6] + v3[5, 7] + v3[5, 8] + v3[5, 9] + v3[5, 10] + v3[5, 11] + v3[5, 12] + v3[5, 13] + v3[5, 14] + v3[5, 15] + v3[5, 16] + v3[5, 17] + v3[5, 18] + v3[5, 19] + v3[5, 20] + v3[5, 21] + v3[5, 22] + v3[5, 23] + v3[5, 24] + v3[5, 25] + v3[5, 26] + v3[5, 27];
    v4[6] := v2[6] + v3[6, 0] + v3[6, 1] + v3[6, 2] + v3[6, 3] + v3[6, 4] + v3[6, 5] + v3[6, 6] + v3[6, 7] + v3[6, 8] + v3[6, 9] + v3[6, 10] + v3[6, 11] + v3[6, 12] + v3[6, 13] + v3[6, 14] + v3[6, 15] + v3[6, 16] + v3[6, 17] + v3[6, 18] + v3[6, 19] + v3[6, 20] + v3[6, 21] + v3[6, 22] + v3[6, 23] + v3[6, 24] + v3[6, 25] + v3[6, 26] + v3[6, 27];
    v4[7] := v2[7] + v3[7, 0] + v3[7, 1] + v3[7, 2] + v3[7, 3] + v3[7, 4] + v3[7, 5] + v3[7, 6] + v3[7, 7] + v3[7, 8] + v3[7, 9] + v3[7, 10] + v3[7, 11] + v3[7, 12] + v3[7, 13] + v3[7, 14] + v3[7, 15] + v3[7, 16] + v3[7, 17] + v3[7, 18] + v3[7, 19] + v3[7, 20] + v3[7, 21] + v3[7, 22] + v3[7, 23] + v3[7, 24] + v3[7, 25] + v3[7, 26] + v3[7, 27];
    v4[8] := v2[8] + v3[8, 0] + v3[8, 1] + v3[8, 2] + v3[8, 3] + v3[8, 4] + v3[8, 5] + v3[8, 6] + v3[8, 7] + v3[8, 8] + v3[8, 9] + v3[8, 10] + v3[8, 11] + v3[8, 12] + v3[8, 13] + v3[8, 14] + v3[8, 15] + v3[8, 16] + v3[8, 17] + v3[8, 18] + v3[8, 19] + v3[8, 20] + v3[8, 21] + v3[8, 22] + v3[8, 23] + v3[8, 24] + v3[8, 25] + v3[8, 26] + v3[8, 27];
    v4[9] := v2[9] + v3[9, 0] + v3[9, 1] + v3[9, 2] + v3[9, 3] + v3[9, 4] + v3[9, 5] + v3[9, 6] + v3[9, 7] + v3[9, 8] + v3[9, 9] + v3[9, 10] + v3[9, 11] + v3[9, 12] + v3[9, 13] + v3[9, 14] + v3[9, 15] + v3[9, 16] + v3[9, 17] + v3[9, 18] + v3[9, 19] + v3[9, 20] + v3[9, 21] + v3[9, 22] + v3[9, 23] + v3[9, 24] + v3[9, 25] + v3[9, 26] + v3[9, 27];
    v4[10] := v2[10] + v3[10, 0] + v3[10, 1] + v3[10, 2] + v3[10, 3] + v3[10, 4] + v3[10, 5] + v3[10, 6] + v3[10, 7] + v3[10, 8] + v3[10, 9] + v3[10, 10] + v3[10, 11] + v3[10, 12] + v3[10, 13] + v3[10, 14] + v3[10, 15] + v3[10, 16] + v3[10, 17] + v3[10, 18] + v3[10, 19] + v3[10, 20] + v3[10, 21] + v3[10, 22] + v3[10, 23] + v3[10, 24] + v3[10, 25] + v3[10, 26] + v3[10, 27];
    v4[11] := v2[11] + v3[11, 0] + v3[11, 1] + v3[11, 2] + v3[11, 3] + v3[11, 4] + v3[11, 5] + v3[11, 6] + v3[11, 7] + v3[11, 8] + v3[11, 9] + v3[11, 10] + v3[11, 11] + v3[11, 12] + v3[11, 13] + v3[11, 14] + v3[11, 15] + v3[11, 16] + v3[11, 17] + v3[11, 18] + v3[11, 19] + v3[11, 20] + v3[11, 21] + v3[11, 22] + v3[11, 23] + v3[11, 24] + v3[11, 25] + v3[11, 26] + v3[11, 27];
    v4[12] := v2[12] + v3[12, 0] + v3[12, 1] + v3[12, 2] + v3[12, 3] + v3[12, 4] + v3[12, 5] + v3[12, 6] + v3[12, 7] + v3[12, 8] + v3[12, 9] + v3[12, 10] + v3[12, 11] + v3[12, 12] + v3[12, 13] + v3[12, 14] + v3[12, 15] + v3[12, 16] + v3[12, 17] + v3[12, 18] + v3[12, 19] + v3[12, 20] + v3[12, 21] + v3[12, 22] + v3[12, 23] + v3[12, 24] + v3[12, 25] + v3[12, 26] + v3[12, 27];
    v4[13] := v2[13] + v3[13, 0] + v3[13, 1] + v3[13, 2] + v3[13, 3] + v3[13, 4] + v3[13, 5] + v3[13, 6] + v3[13, 7] + v3[13, 8] + v3[13, 9] + v3[13, 10] + v3[13, 11] + v3[13, 12] + v3[13, 13] + v3[13, 14] + v3[13, 15] + v3[13, 16] + v3[13, 17] + v3[13, 18] + v3[13, 19] + v3[13, 20] + v3[13, 21] + v3[13, 22] + v3[13, 23] + v3[13, 24] + v3[13, 25] + v3[13, 26] + v3[13, 27];
    v4[14] := v2[14] + v3[14, 0] + v3[14, 1] + v3[14, 2] + v3[14, 3] + v3[14, 4] + v3[14, 5] + v3[14, 6] + v3[14, 7] + v3[14, 8] + v3[14, 9] + v3[14, 10] + v3[14, 11] + v3[14, 12] + v3[14, 13] + v3[14, 14] + v3[14, 15] + v3[14, 16] + v3[14, 17] + v3[14, 18] + v3[14, 19] + v3[14, 20] + v3[14, 21] + v3[14, 22] + v3[14, 23] + v3[14, 24] + v3[14, 25] + v3[14, 26] + v3[14, 27];
    v4[15] := v2[15] + v3[15, 0] + v3[15, 1] + v3[15, 2] + v3[15, 3] + v3[15, 4] + v3[15, 5] + v3[15, 6] + v3[15, 7] + v3[15, 8] + v3[15, 9] + v3[15, 10] + v3[15, 11] + v3[15, 12] + v3[15, 13] + v3[15, 14] + v3[15, 15] + v3[15, 16] + v3[15, 17] + v3[15, 18] + v3[15, 19] + v3[15, 20] + v3[15, 21] + v3[15, 22] + v3[15, 23] + v3[15, 24] + v3[15, 25] + v3[15, 26] + v3[15, 27];

    // ---- l1_silu: SILU ----
    v5[0] := v4[0] / (1.0 + EXP(-v4[0]));
    v5[1] := v4[1] / (1.0 + EXP(-v4[1]));
    v5[2] := v4[2] / (1.0 + EXP(-v4[2]));
    v5[3] := v4[3] / (1.0 + EXP(-v4[3]));
    v5[4] := v4[4] / (1.0 + EXP(-v4[4]));
    v5[5] := v4[5] / (1.0 + EXP(-v4[5]));
    v5[6] := v4[6] / (1.0 + EXP(-v4[6]));
    v5[7] := v4[7] / (1.0 + EXP(-v4[7]));
    v5[8] := v4[8] / (1.0 + EXP(-v4[8]));
    v5[9] := v4[9] / (1.0 + EXP(-v4[9]));
    v5[10] := v4[10] / (1.0 + EXP(-v4[10]));
    v5[11] := v4[11] / (1.0 + EXP(-v4[11]));
    v5[12] := v4[12] / (1.0 + EXP(-v4[12]));
    v5[13] := v4[13] / (1.0 + EXP(-v4[13]));
    v5[14] := v4[14] / (1.0 + EXP(-v4[14]));
    v5[15] := v4[15] / (1.0 + EXP(-v4[15]));

    // ---- l1_bspline: BsplineLUT(16x4, 15pts) HOISTED ----
    // Binary search ONCE per input, shared across outputs
    // --- Input 0: binary search ---
    lo := 0; hi := 14;
    WHILE hi - lo > 1 DO
        mid := lo + (hi - lo) / 2;
        IF v4[0] > "NeuroPLC_Weights".w3[mid] THEN lo := mid; ELSE hi := mid; END_IF;
    END_WHILE;
    t_val := (v4[0] - "NeuroPLC_Weights".w3[lo]) / ("NeuroPLC_Weights".w3[hi] - "NeuroPLC_Weights".w3[lo] + 1.0E-10);
    v7[0, 0] := "NeuroPLC_Weights".w4[0 + lo] * (1.0 - t_val) + "NeuroPLC_Weights".w4[0 + hi] * t_val;
    v7[1, 0] := "NeuroPLC_Weights".w4[240 + lo] * (1.0 - t_val) + "NeuroPLC_Weights".w4[240 + hi] * t_val;
    v7[2, 0] := "NeuroPLC_Weights".w4[480 + lo] * (1.0 - t_val) + "NeuroPLC_Weights".w4[480 + hi] * t_val;
    v7[3, 0] := "NeuroPLC_Weights".w4[720 + lo] * (1.0 - t_val) + "NeuroPLC_Weights".w4[720 + hi] * t_val;

    // --- Input 1: binary search ---
    lo := 0; hi := 14;
    WHILE hi - lo > 1 DO
        mid := lo + (hi - lo) / 2;
        IF v4[1] > "NeuroPLC_Weights".w3[mid] THEN lo := mid; ELSE hi := mid; END_IF;
    END_WHILE;
    t_val := (v4[1] - "NeuroPLC_Weights".w3[lo]) / ("NeuroPLC_Weights".w3[hi] - "NeuroPLC_Weights".w3[lo] + 1.0E-10);
    v7[0, 1] := "NeuroPLC_Weights".w4[15 + lo] * (1.0 - t_val) + "NeuroPLC_Weights".w4[15 + hi] * t_val;
    v7[1, 1] := "NeuroPLC_Weights".w4[255 + lo] * (1.0 - t_val) + "NeuroPLC_Weights".w4[255 + hi] * t_val;
    v7[2, 1] := "NeuroPLC_Weights".w4[495 + lo] * (1.0 - t_val) + "NeuroPLC_Weights".w4[495 + hi] * t_val;
    v7[3, 1] := "NeuroPLC_Weights".w4[735 + lo] * (1.0 - t_val) + "NeuroPLC_Weights".w4[735 + hi] * t_val;

    // --- Input 2: binary search ---
    lo := 0; hi := 14;
    WHILE hi - lo > 1 DO
        mid := lo + (hi - lo) / 2;
        IF v4[2] > "NeuroPLC_Weights".w3[mid] THEN lo := mid; ELSE hi := mid; END_IF;
    END_WHILE;
    t_val := (v4[2] - "NeuroPLC_Weights".w3[lo]) / ("NeuroPLC_Weights".w3[hi] - "NeuroPLC_Weights".w3[lo] + 1.0E-10);
    v7[0, 2] := "NeuroPLC_Weights".w4[30 + lo] * (1.0 - t_val) + "NeuroPLC_Weights".w4[30 + hi] * t_val;
    v7[1, 2] := "NeuroPLC_Weights".w4[270 + lo] * (1.0 - t_val) + "NeuroPLC_Weights".w4[270 + hi] * t_val;
    v7[2, 2] := "NeuroPLC_Weights".w4[510 + lo] * (1.0 - t_val) + "NeuroPLC_Weights".w4[510 + hi] * t_val;
    v7[3, 2] := "NeuroPLC_Weights".w4[750 + lo] * (1.0 - t_val) + "NeuroPLC_Weights".w4[750 + hi] * t_val;

    // --- Input 3: binary search ---
    lo := 0; hi := 14;
    WHILE hi - lo > 1 DO
        mid := lo + (hi - lo) / 2;
        IF v4[3] > "NeuroPLC_Weights".w3[mid] THEN lo := mid; ELSE hi := mid; END_IF;
    END_WHILE;
    t_val := (v4[3] - "NeuroPLC_Weights".w3[lo]) / ("NeuroPLC_Weights".w3[hi] - "NeuroPLC_Weights".w3[lo] + 1.0E-10);
    v7[0, 3] := "NeuroPLC_Weights".w4[45 + lo] * (1.0 - t_val) + "NeuroPLC_Weights".w4[45 + hi] * t_val;
    v7[1, 3] := "NeuroPLC_Weights".w4[285 + lo] * (1.0 - t_val) + "NeuroPLC_Weights".w4[285 + hi] * t_val;
    v7[2, 3] := "NeuroPLC_Weights".w4[525 + lo] * (1.0 - t_val) + "NeuroPLC_Weights".w4[525 + hi] * t_val;
    v7[3, 3] := "NeuroPLC_Weights".w4[765 + lo] * (1.0 - t_val) + "NeuroPLC_Weights".w4[765 + hi] * t_val;

    // --- Input 4: binary search ---
    lo := 0; hi := 14;
    WHILE hi - lo > 1 DO
        mid := lo + (hi - lo) / 2;
        IF v4[4] > "NeuroPLC_Weights".w3[mid] THEN lo := mid; ELSE hi := mid; END_IF;
    END_WHILE;
    t_val := (v4[4] - "NeuroPLC_Weights".w3[lo]) / ("NeuroPLC_Weights".w3[hi] - "NeuroPLC_Weights".w3[lo] + 1.0E-10);
    v7[0, 4] := "NeuroPLC_Weights".w4[60 + lo] * (1.0 - t_val) + "NeuroPLC_Weights".w4[60 + hi] * t_val;
    v7[1, 4] := "NeuroPLC_Weights".w4[300 + lo] * (1.0 - t_val) + "NeuroPLC_Weights".w4[300 + hi] * t_val;
    v7[2, 4] := "NeuroPLC_Weights".w4[540 + lo] * (1.0 - t_val) + "NeuroPLC_Weights".w4[540 + hi] * t_val;
    v7[3, 4] := "NeuroPLC_Weights".w4[780 + lo] * (1.0 - t_val) + "NeuroPLC_Weights".w4[780 + hi] * t_val;

    // --- Input 5: binary search ---
    lo := 0; hi := 14;
    WHILE hi - lo > 1 DO
        mid := lo + (hi - lo) / 2;
        IF v4[5] > "NeuroPLC_Weights".w3[mid] THEN lo := mid; ELSE hi := mid; END_IF;
    END_WHILE;
    t_val := (v4[5] - "NeuroPLC_Weights".w3[lo]) / ("NeuroPLC_Weights".w3[hi] - "NeuroPLC_Weights".w3[lo] + 1.0E-10);
    v7[0, 5] := "NeuroPLC_Weights".w4[75 + lo] * (1.0 - t_val) + "NeuroPLC_Weights".w4[75 + hi] * t_val;
    v7[1, 5] := "NeuroPLC_Weights".w4[315 + lo] * (1.0 - t_val) + "NeuroPLC_Weights".w4[315 + hi] * t_val;
    v7[2, 5] := "NeuroPLC_Weights".w4[555 + lo] * (1.0 - t_val) + "NeuroPLC_Weights".w4[555 + hi] * t_val;
    v7[3, 5] := "NeuroPLC_Weights".w4[795 + lo] * (1.0 - t_val) + "NeuroPLC_Weights".w4[795 + hi] * t_val;

    // --- Input 6: binary search ---
    lo := 0; hi := 14;
    WHILE hi - lo > 1 DO
        mid := lo + (hi - lo) / 2;
        IF v4[6] > "NeuroPLC_Weights".w3[mid] THEN lo := mid; ELSE hi := mid; END_IF;
    END_WHILE;
    t_val := (v4[6] - "NeuroPLC_Weights".w3[lo]) / ("NeuroPLC_Weights".w3[hi] - "NeuroPLC_Weights".w3[lo] + 1.0E-10);
    v7[0, 6] := "NeuroPLC_Weights".w4[90 + lo] * (1.0 - t_val) + "NeuroPLC_Weights".w4[90 + hi] * t_val;
    v7[1, 6] := "NeuroPLC_Weights".w4[330 + lo] * (1.0 - t_val) + "NeuroPLC_Weights".w4[330 + hi] * t_val;
    v7[2, 6] := "NeuroPLC_Weights".w4[570 + lo] * (1.0 - t_val) + "NeuroPLC_Weights".w4[570 + hi] * t_val;
    v7[3, 6] := "NeuroPLC_Weights".w4[810 + lo] * (1.0 - t_val) + "NeuroPLC_Weights".w4[810 + hi] * t_val;

    // --- Input 7: binary search ---
    lo := 0; hi := 14;
    WHILE hi - lo > 1 DO
        mid := lo + (hi - lo) / 2;
        IF v4[7] > "NeuroPLC_Weights".w3[mid] THEN lo := mid; ELSE hi := mid; END_IF;
    END_WHILE;
    t_val := (v4[7] - "NeuroPLC_Weights".w3[lo]) / ("NeuroPLC_Weights".w3[hi] - "NeuroPLC_Weights".w3[lo] + 1.0E-10);
    v7[0, 7] := "NeuroPLC_Weights".w4[105 + lo] * (1.0 - t_val) + "NeuroPLC_Weights".w4[105 + hi] * t_val;
    v7[1, 7] := "NeuroPLC_Weights".w4[345 + lo] * (1.0 - t_val) + "NeuroPLC_Weights".w4[345 + hi] * t_val;
    v7[2, 7] := "NeuroPLC_Weights".w4[585 + lo] * (1.0 - t_val) + "NeuroPLC_Weights".w4[585 + hi] * t_val;
    v7[3, 7] := "NeuroPLC_Weights".w4[825 + lo] * (1.0 - t_val) + "NeuroPLC_Weights".w4[825 + hi] * t_val;

    // --- Input 8: binary search ---
    lo := 0; hi := 14;
    WHILE hi - lo > 1 DO
        mid := lo + (hi - lo) / 2;
        IF v4[8] > "NeuroPLC_Weights".w3[mid] THEN lo := mid; ELSE hi := mid; END_IF;
    END_WHILE;
    t_val := (v4[8] - "NeuroPLC_Weights".w3[lo]) / ("NeuroPLC_Weights".w3[hi] - "NeuroPLC_Weights".w3[lo] + 1.0E-10);
    v7[0, 8] := "NeuroPLC_Weights".w4[120 + lo] * (1.0 - t_val) + "NeuroPLC_Weights".w4[120 + hi] * t_val;
    v7[1, 8] := "NeuroPLC_Weights".w4[360 + lo] * (1.0 - t_val) + "NeuroPLC_Weights".w4[360 + hi] * t_val;
    v7[2, 8] := "NeuroPLC_Weights".w4[600 + lo] * (1.0 - t_val) + "NeuroPLC_Weights".w4[600 + hi] * t_val;
    v7[3, 8] := "NeuroPLC_Weights".w4[840 + lo] * (1.0 - t_val) + "NeuroPLC_Weights".w4[840 + hi] * t_val;

    // --- Input 9: binary search ---
    lo := 0; hi := 14;
    WHILE hi - lo > 1 DO
        mid := lo + (hi - lo) / 2;
        IF v4[9] > "NeuroPLC_Weights".w3[mid] THEN lo := mid; ELSE hi := mid; END_IF;
    END_WHILE;
    t_val := (v4[9] - "NeuroPLC_Weights".w3[lo]) / ("NeuroPLC_Weights".w3[hi] - "NeuroPLC_Weights".w3[lo] + 1.0E-10);
    v7[0, 9] := "NeuroPLC_Weights".w4[135 + lo] * (1.0 - t_val) + "NeuroPLC_Weights".w4[135 + hi] * t_val;
    v7[1, 9] := "NeuroPLC_Weights".w4[375 + lo] * (1.0 - t_val) + "NeuroPLC_Weights".w4[375 + hi] * t_val;
    v7[2, 9] := "NeuroPLC_Weights".w4[615 + lo] * (1.0 - t_val) + "NeuroPLC_Weights".w4[615 + hi] * t_val;
    v7[3, 9] := "NeuroPLC_Weights".w4[855 + lo] * (1.0 - t_val) + "NeuroPLC_Weights".w4[855 + hi] * t_val;

    // --- Input 10: binary search ---
    lo := 0; hi := 14;
    WHILE hi - lo > 1 DO
        mid := lo + (hi - lo) / 2;
        IF v4[10] > "NeuroPLC_Weights".w3[mid] THEN lo := mid; ELSE hi := mid; END_IF;
    END_WHILE;
    t_val := (v4[10] - "NeuroPLC_Weights".w3[lo]) / ("NeuroPLC_Weights".w3[hi] - "NeuroPLC_Weights".w3[lo] + 1.0E-10);
    v7[0, 10] := "NeuroPLC_Weights".w4[150 + lo] * (1.0 - t_val) + "NeuroPLC_Weights".w4[150 + hi] * t_val;
    v7[1, 10] := "NeuroPLC_Weights".w4[390 + lo] * (1.0 - t_val) + "NeuroPLC_Weights".w4[390 + hi] * t_val;
    v7[2, 10] := "NeuroPLC_Weights".w4[630 + lo] * (1.0 - t_val) + "NeuroPLC_Weights".w4[630 + hi] * t_val;
    v7[3, 10] := "NeuroPLC_Weights".w4[870 + lo] * (1.0 - t_val) + "NeuroPLC_Weights".w4[870 + hi] * t_val;

    // --- Input 11: binary search ---
    lo := 0; hi := 14;
    WHILE hi - lo > 1 DO
        mid := lo + (hi - lo) / 2;
        IF v4[11] > "NeuroPLC_Weights".w3[mid] THEN lo := mid; ELSE hi := mid; END_IF;
    END_WHILE;
    t_val := (v4[11] - "NeuroPLC_Weights".w3[lo]) / ("NeuroPLC_Weights".w3[hi] - "NeuroPLC_Weights".w3[lo] + 1.0E-10);
    v7[0, 11] := "NeuroPLC_Weights".w4[165 + lo] * (1.0 - t_val) + "NeuroPLC_Weights".w4[165 + hi] * t_val;
    v7[1, 11] := "NeuroPLC_Weights".w4[405 + lo] * (1.0 - t_val) + "NeuroPLC_Weights".w4[405 + hi] * t_val;
    v7[2, 11] := "NeuroPLC_Weights".w4[645 + lo] * (1.0 - t_val) + "NeuroPLC_Weights".w4[645 + hi] * t_val;
    v7[3, 11] := "NeuroPLC_Weights".w4[885 + lo] * (1.0 - t_val) + "NeuroPLC_Weights".w4[885 + hi] * t_val;

    // --- Input 12: binary search ---
    lo := 0; hi := 14;
    WHILE hi - lo > 1 DO
        mid := lo + (hi - lo) / 2;
        IF v4[12] > "NeuroPLC_Weights".w3[mid] THEN lo := mid; ELSE hi := mid; END_IF;
    END_WHILE;
    t_val := (v4[12] - "NeuroPLC_Weights".w3[lo]) / ("NeuroPLC_Weights".w3[hi] - "NeuroPLC_Weights".w3[lo] + 1.0E-10);
    v7[0, 12] := "NeuroPLC_Weights".w4[180 + lo] * (1.0 - t_val) + "NeuroPLC_Weights".w4[180 + hi] * t_val;
    v7[1, 12] := "NeuroPLC_Weights".w4[420 + lo] * (1.0 - t_val) + "NeuroPLC_Weights".w4[420 + hi] * t_val;
    v7[2, 12] := "NeuroPLC_Weights".w4[660 + lo] * (1.0 - t_val) + "NeuroPLC_Weights".w4[660 + hi] * t_val;
    v7[3, 12] := "NeuroPLC_Weights".w4[900 + lo] * (1.0 - t_val) + "NeuroPLC_Weights".w4[900 + hi] * t_val;

    // --- Input 13: binary search ---
    lo := 0; hi := 14;
    WHILE hi - lo > 1 DO
        mid := lo + (hi - lo) / 2;
        IF v4[13] > "NeuroPLC_Weights".w3[mid] THEN lo := mid; ELSE hi := mid; END_IF;
    END_WHILE;
    t_val := (v4[13] - "NeuroPLC_Weights".w3[lo]) / ("NeuroPLC_Weights".w3[hi] - "NeuroPLC_Weights".w3[lo] + 1.0E-10);
    v7[0, 13] := "NeuroPLC_Weights".w4[195 + lo] * (1.0 - t_val) + "NeuroPLC_Weights".w4[195 + hi] * t_val;
    v7[1, 13] := "NeuroPLC_Weights".w4[435 + lo] * (1.0 - t_val) + "NeuroPLC_Weights".w4[435 + hi] * t_val;
    v7[2, 13] := "NeuroPLC_Weights".w4[675 + lo] * (1.0 - t_val) + "NeuroPLC_Weights".w4[675 + hi] * t_val;
    v7[3, 13] := "NeuroPLC_Weights".w4[915 + lo] * (1.0 - t_val) + "NeuroPLC_Weights".w4[915 + hi] * t_val;

    // --- Input 14: binary search ---
    lo := 0; hi := 14;
    WHILE hi - lo > 1 DO
        mid := lo + (hi - lo) / 2;
        IF v4[14] > "NeuroPLC_Weights".w3[mid] THEN lo := mid; ELSE hi := mid; END_IF;
    END_WHILE;
    t_val := (v4[14] - "NeuroPLC_Weights".w3[lo]) / ("NeuroPLC_Weights".w3[hi] - "NeuroPLC_Weights".w3[lo] + 1.0E-10);
    v7[0, 14] := "NeuroPLC_Weights".w4[210 + lo] * (1.0 - t_val) + "NeuroPLC_Weights".w4[210 + hi] * t_val;
    v7[1, 14] := "NeuroPLC_Weights".w4[450 + lo] * (1.0 - t_val) + "NeuroPLC_Weights".w4[450 + hi] * t_val;
    v7[2, 14] := "NeuroPLC_Weights".w4[690 + lo] * (1.0 - t_val) + "NeuroPLC_Weights".w4[690 + hi] * t_val;
    v7[3, 14] := "NeuroPLC_Weights".w4[930 + lo] * (1.0 - t_val) + "NeuroPLC_Weights".w4[930 + hi] * t_val;

    // --- Input 15: binary search ---
    lo := 0; hi := 14;
    WHILE hi - lo > 1 DO
        mid := lo + (hi - lo) / 2;
        IF v4[15] > "NeuroPLC_Weights".w3[mid] THEN lo := mid; ELSE hi := mid; END_IF;
    END_WHILE;
    t_val := (v4[15] - "NeuroPLC_Weights".w3[lo]) / ("NeuroPLC_Weights".w3[hi] - "NeuroPLC_Weights".w3[lo] + 1.0E-10);
    v7[0, 15] := "NeuroPLC_Weights".w4[225 + lo] * (1.0 - t_val) + "NeuroPLC_Weights".w4[225 + hi] * t_val;
    v7[1, 15] := "NeuroPLC_Weights".w4[465 + lo] * (1.0 - t_val) + "NeuroPLC_Weights".w4[465 + hi] * t_val;
    v7[2, 15] := "NeuroPLC_Weights".w4[705 + lo] * (1.0 - t_val) + "NeuroPLC_Weights".w4[705 + hi] * t_val;
    v7[3, 15] := "NeuroPLC_Weights".w4[945 + lo] * (1.0 - t_val) + "NeuroPLC_Weights".w4[945 + hi] * t_val;


    // ---- l1_base: MatMul(16→4) ----
    // W = "NeuroPLC_Weights".w5[:64],   b = w5[64:]
    v6[0] := "NeuroPLC_Weights".w5[64 + 0];
    FOR i := 0 TO 15 DO
        v6[0] := v6[0] + "NeuroPLC_Weights".w5[0 + i] * v5[i];
    END_FOR;
    v6[1] := "NeuroPLC_Weights".w5[64 + 1];
    FOR i := 0 TO 15 DO
        v6[1] := v6[1] + "NeuroPLC_Weights".w5[16 + i] * v5[i];
    END_FOR;
    v6[2] := "NeuroPLC_Weights".w5[64 + 2];
    FOR i := 0 TO 15 DO
        v6[2] := v6[2] + "NeuroPLC_Weights".w5[32 + i] * v5[i];
    END_FOR;
    v6[3] := "NeuroPLC_Weights".w5[64 + 3];
    FOR i := 0 TO 15 DO
        v6[3] := v6[3] + "NeuroPLC_Weights".w5[48 + i] * v5[i];
    END_FOR;

    // ---- l1_merge: Add (KAN merge) ----
    v8[0] := v6[0] + v7[0, 0] + v7[0, 1] + v7[0, 2] + v7[0, 3] + v7[0, 4] + v7[0, 5] + v7[0, 6] + v7[0, 7] + v7[0, 8] + v7[0, 9] + v7[0, 10] + v7[0, 11] + v7[0, 12] + v7[0, 13] + v7[0, 14] + v7[0, 15];
    v8[1] := v6[1] + v7[1, 0] + v7[1, 1] + v7[1, 2] + v7[1, 3] + v7[1, 4] + v7[1, 5] + v7[1, 6] + v7[1, 7] + v7[1, 8] + v7[1, 9] + v7[1, 10] + v7[1, 11] + v7[1, 12] + v7[1, 13] + v7[1, 14] + v7[1, 15];
    v8[2] := v6[2] + v7[2, 0] + v7[2, 1] + v7[2, 2] + v7[2, 3] + v7[2, 4] + v7[2, 5] + v7[2, 6] + v7[2, 7] + v7[2, 8] + v7[2, 9] + v7[2, 10] + v7[2, 11] + v7[2, 12] + v7[2, 13] + v7[2, 14] + v7[2, 15];
    v8[3] := v6[3] + v7[3, 0] + v7[3, 1] + v7[3, 2] + v7[3, 3] + v7[3, 4] + v7[3, 5] + v7[3, 6] + v7[3, 7] + v7[3, 8] + v7[3, 9] + v7[3, 10] + v7[3, 11] + v7[3, 12] + v7[3, 13] + v7[3, 14] + v7[3, 15];

    // ---- softmax: Softmax ----
    v9[0] := EXP(v8[0]);
    v9[1] := EXP(v8[1]);
    v9[2] := EXP(v8[2]);
    v9[3] := EXP(v8[3]);
    sum_val := v9[0]
             + v9[1]
             + v9[2]
             + v9[3]
             ;
    IF sum_val > 0.0 THEN
        v9[0] := v9[0] / sum_val;
        v9[1] := v9[1] / sum_val;
        v9[2] := v9[2] / sum_val;
        v9[3] := v9[3] / sum_val;
    END_IF;

    // ---- Argmax ----
    max_val := v10[0];
    fault_class := 0;
    IF v10[1] > max_val THEN
        max_val := v10[1];
        fault_class := 1;
    END_IF;
    IF v10[2] > max_val THEN
        max_val := v10[2];
        fault_class := 2;
    END_IF;
    IF v10[3] > max_val THEN
        max_val := v10[3];
        fault_class := 3;
    END_IF;
    confidence := max_val;

END_FUNCTION_BLOCK